// TwinCAT 3 PLC project OP710_Robotic_Weld
// ProgramVersion: 3.1.4024.0
// libraries:
//   Tc2_Standard, * (Beckhoff Automation GmbH)
//   Tc2_System, * (Beckhoff Automation GmbH)
//   Tc3_Module, * (Beckhoff Automation GmbH)
//   VisuDialogs, * (System)
// project tree:
//   DUTs/ Fixture.TcDUT, MH_Robot.TcDUT, Weld_Robot.TcDUT
//   / GlobalTextList.TcGTLO, PlcTask.TcTTO, Visualization Manager.TcVMO (not stored)
//   GVLs/ Inputs.TcGVL, Memory.TcGVL, Outputs.TcGVL
//   POUs/ Auto_Cycle_Fix1.TcPOU, Auto_Cycle_Fix2.TcPOU, Fix1_FB.TcPOU, Fix2_FB.TcPOU, MAIN.TcPOU, Robot_MH.TcPOU, Robot_Weld.TcPOU, RollerDoor.TcPOU, Trunnion.TcPOU, TurnTable.TcPOU
//   VISUs/ Auto_Cycle_Fix1.TcVIS, Auto_Cycle_Fix2.TcVIS, Manual_Action_Fix1.TcVIS, Manual_Action_Fix2.TcVIS
// real-time tasks:
//   TASK PlcTask: cycle T#10ms, priority 20, ADS port 350

CONFIGURATION OP710_Robotic_Weld
    RESOURCE PLC ON TwinCAT3
        TASK PlcTask(INTERVAL := T#10ms, PRIORITY := 20);
        PROGRAM MAIN WITH PlcTask : MAIN;
    END_RESOURCE
END_CONFIGURATION

// ---- DUTs/Fixture.TcDUT
TYPE Fixture :
STRUCT
	i_Clamp1_Fbk : BOOL;
	i_Clamp2_Fbk : BOOL;
	i_Clamp3_Fbk : BOOL;
	
	i_Declamp1_Fbk : BOOL;
	i_Declamp2_Fbk : BOOL;
	i_Declamp3_Fbk : BOOL;
	
	o_Clamp_HP : BOOL;
	o_Clamp_WP : BOOL;
	
	Work_Position : BOOL;
	Home_Position : BOOL;
	Manual_Sel : BOOL;
	Auto_Sel : BOOL;
	
END_STRUCT
END_TYPE

// ---- DUTs/MH_Robot.TcDUT
TYPE MH_Robot :
STRUCT
	i_Home 			: BOOL;
	i_Prg_No		: INT;
	i_Start			: BOOL;	
	i_Area_Ok1		: BOOL;
	i_Area_Ok2		: BOOL;
	
	o_Pickup_Comp1	: BOOL;
	o_Pickup_Comp2	: BOOL;
		
END_STRUCT
END_TYPE

// ---- DUTs/Weld_Robot.TcDUT
TYPE Weld_Robot :
STRUCT
	i_Home 		: BOOL;
	i_Prg_No	: INT;
	i_Start		: BOOL;	
	i_Area_Ok	: BOOL;
	
	o_Weld_Comp	: BOOL;
	
END_STRUCT
END_TYPE

// ---- GVLs/Inputs.TcGVL

//(------INPUTS--------)

VAR_GLOBAL
	
i_Control_Pressure_Sw_In1_BPB1 AT %IX0.0 : BOOL;	//Control Pressure Switch Input 1-BPB1  
i_Control_Pressure_Sw_In2_BPB1 AT %IX0.1 : BOOL;	//Control Pressure Switch Input 2-BPB1  
i_Valve_Pos_BGB1 AT %IX0.2 : BOOL;					//Valve Position-BGB1
i_CC6_Clamp_1_Sensor_HP AT %IX0.4 : BOOL;			//Clamping Circuit 6 Clamping Unit 1 sensor  HP
i_CC6_Clamp_1_Sensor_WP AT %IX0.5 : BOOL;			//Clamping Circuit 6 Clamping Unit 1 sensor  WP
i_CC4_Clamp_3_Sensor_HP AT %IX0.6 : BOOL;			//Clamping Circuit 4 Clamping Unit 3 sensor  HP
i_CC4_Clamp_3_Sensor_WP AT %IX0.7 : BOOL;			//Clamping Circuit 4 Clamping Unit 3 sensor  WP
i_PART_CONTROL_B13 AT %IX1.0 : BOOL;				//PART CONTROL  B13
i_PART_CONTROL_B27 AT %IX1.1 : BOOL;				//PART CONTROL  B27
i_PART_CONTROL_B14 AT %IX1.2 : BOOL;				//PART CONTROL  B14
i_PART_CONTROL_B28 AT %IX1.3 : BOOL;				//PART CONTROL  B28
i_KEC6_Slave_module_1_2_1 AT %IX1.6 : BOOL;			//Connect to KEC6 Salve module 1.2
i_KEC6_Slave_module_1_2_2 AT %IX1.7 : BOOL;			//Connect to KEC6 Salve module 1.2

i_CC4_Clamp_2_Sensor_HP	AT %IX4.0 : BOOL;			//Clamping Circuit 4 Clamping Unit 2 sensor HP
i_CC4_Clamp_2_Sensor_WP	AT %IX4.1 : BOOL;			//Clamping Circuit 4 Clamping Unit 2 sensor WP
i_CC4_Clamp_1_Sensor_HP	AT %IX4.2 : BOOL;			//Clamping Circuit 4 Clamping Unit 1 sensor HP
i_CC4_Clamp_1_Sensor_WP	AT %IX4.3 : BOOL;			//Clamping Circuit 4 Clamping Unit 1 sensor WP
i_CC2_Clamp_3_Sensor_HP	AT %IX4.4 : BOOL;			//Clamping Circuit 2 Clamping Unit 3 sensor HP
i_CC2_Clamp_3_Sensor_WP	AT %IX4.5 : BOOL;			//Clamping Circuit 2 Clamping Unit 3 sensor WP
i_PART_CONTROL_B12	AT %IX4.6 : BOOL;				//PART CONTROL B12
i_PART_CONTROL_B26	AT %IX4.7 : BOOL;				//PART CONTROL B26

i_PART_CONTROL_B11	AT %IX5.0 : BOOL;				//PART CONTROL B11
i_PART_CONTROL_B25	AT %IX5.1 : BOOL;				//PART CONTROL B25
i_PART_CONTROL_B10	AT %IX5.2 : BOOL;				//PART CONTROL B10
i_PART_CONTROL_B24	AT %IX5.3 : BOOL;				//PART CONTROL B24

i_CC3_Clamp_3_Sensor_HP AT %IX8.0 : BOOL;			//Clamping Circuit 3 Clamping Unit 3 sensor HP
i_CC3_Clamp_3_Sensor_WP AT %IX8.1 : BOOL;			//Clamping Circuit 3 Clamping Unit 3 sensor WP
i_CC3_Clamp_2_Sensor_HP AT %IX8.2 : BOOL;			//Clamping Circuit 3 Clamping Unit 2 sensor HP
i_CC3_Clamp_2_Sensor_WP AT %IX8.3 : BOOL;			//Clamping Circuit 3 Clamping Unit 2 sensor WP
i_CC3_Clamp_1_Sensor_HP AT %IX8.4 : BOOL;			//Clamping Circuit 3 Clamping Unit 1 sensor HP
i_CC3_Clamp_1_Sensor_WP AT %IX8.5 : BOOL;			//Clamping Circuit 3 Clamping Unit 1 sensor WP
i_PART_CONTROL_B7 AT %IX8.6 : BOOL;					//PART CONTROL B7
i_PART_CONTROL_B21 AT %IX8.7 : BOOL;				//PART CONTROL B21

i_PART_CONTROL_B6 AT %IX9.0 : BOOL;					//PART CONTROL B6
i_PART_CONTROL_B20 AT %IX9.1 : BOOL;				//PART CONTROL B20
i_PART_CONTROL_B5 AT %IX9.2 : BOOL;					//PART CONTROL B5
i_PART_CONTROL_B19 AT %IX9.3 : BOOL;				//PART CONTROL B19
i_KEC8_Slave_module_2_2_1 AT %IX9.6 : BOOL;			//Connect to KEC8 Salve module 2.2
i_KEC8_Slave_module_2_2_2 AT %IX9.7 : BOOL;			//Connect to KEC8 Salve module 2.2

i_CC1_Clamp_3_Sensor_HP AT %IX12.0 : BOOL;			//Clamping Circuit 1 Clamping Unit 3 sensor HP
i_CC1_Clamp_3_Sensor_WP AT %IX12.1 : BOOL;			//Clamping Circuit 1 Clamping Unit 3 sensor WP
i_CC1_Clamp_2_Sensor_HP AT %IX12.2 : BOOL;			//Clamping Circuit 1 Clamping Unit 2 sensor HP
i_CC1_Clamp_2_Sensor_WP AT %IX12.3 : BOOL;			//Clamping Circuit 1 Clamping Unit 2 sensor WP
i_CC1_Clamp_1_Sensor_HP AT %IX12.4 : BOOL;			//Clamping Circuit 1 Clamping Unit 1 sensor HP
i_CC1_Clamp_1_Sensor_WP AT %IX12.5 : BOOL;			//Clamping Circuit 1 Clamping Unit 1 sensor WP
i_PART_CONTROL_B4 AT %IX12.6 : BOOL;				//PART CONTROL B4
i_PART_CONTROL_B18 AT %IX12.7 : BOOL;				//PART CONTROL B18

i_PART_CONTROL_B3 AT %IX13.0 : BOOL;				//PART CONTROL B3
i_PART_CONTROL_B17 AT %IX13.1 : BOOL;				//PART CONTROL B17
i_PART_CONTROL_B2 AT %IX13.2 : BOOL;				//PART CONTROL B2
i_PART_CONTROL_B16 AT %IX13.3 : BOOL;				//PART CONTROL B16

i_CC2_Clamp_2_Sensor_HP AT %IX16.0 : BOOL;			//Clamping Circuit 2 Clamping Unit 2 sensor HP
i_CC2_Clamp_2_Sensor_WP AT %IX16.1 : BOOL;			//Clamping Circuit 2 Clamping Unit 2 sensor WP
i_CC2_Clamp_1_Sensor_HP AT %IX16.2 : BOOL;			//Clamping Circuit 2 Clamping Unit 1 sensor HP
i_CC2_Clamp_1_Sensor_WP AT %IX16.3 : BOOL;			//Clamping Circuit 2 Clamping Unit 1 sensor WP
i_PART_CONTROL_B9 AT %IX16.4 : BOOL;				//PART CONTROL B9
i_PART_CONTROL_B23 AT %IX16.5 : BOOL;				//PART CONTROL B23
i_PART_CONTROL_B8 AT %IX16.6 : BOOL;				//PART CONTROL B8
i_PART_CONTROL_B22 AT %IX16.7 : BOOL;				//PART CONTROL B22

i_CC5_Clamp_1_Sensor_HP AT %IX24.0 : BOOL;			//Clamping Circuit 5 Clamping Unit 1 sensor HP
i_CC5_Clamp_1_Sensor_WP AT %IX24.1 : BOOL;			//Clamping Circuit 5 Clamping Unit 1 sensor WP
i_PART_CONTROL_B1 AT %IX24.2 : BOOL;				//PART CONTROL B1
i_PART_CONTROL_B15 AT %IX24.3 : BOOL;				//PART CONTROL B15

i_TR_0_Deg AT %I* : BOOL;							//Trunnion at 0 degree
i_TR_20_Degree AT %I* : BOOL;						//Trunnion at -20 degree
i_TR_45_Degree AT %I* : BOOL;						//Trunnion at 45 degree
i_TR_50_Degree AT %I* : BOOL;						//Trunnion at 50 degree
i_TR_80_Degree AT %I* : BOOL;						//Trunnion at 80 degree
i_TT_0_Degree AT %I* : BOOL;
i_TT_180_Degree AT %I* : BOOL;

Roller_Door_Up AT %I* : BOOL;						//Roller Door Up
Roller_Door_Down AT %I* : BOOL;						//Roller Door Down


END_VAR

// ---- GVLs/Memory.TcGVL
VAR_GLOBAL
	
Start_Pb     		: BOOL;						    // Station Cycle Start Pb
Station_Mode 		: INT;							// Station Manual/Auto Pb
Fix_Sel   	 		: INT;							//Station Select Pb, 0 - OP710 Long, 1 - OP710 Short
Auto_Mode	 		: BOOL;
Manual_Mode	 		: BOOL;
Master_On	 		: BOOL;
EStop				: BOOL;
Safety_Ok	 		: BOOL;
Fault_Reset			: BOOL;
Fix1_Part_1_Load  	: BOOL;
Fix1_Part_2_Load  	: BOOL;
Fix2_Part_1_Load  	: BOOL;
Fix2_Part_2_Load  	: BOOL;
Return_Home  		: BOOL;

i_B : ARRAY [0..28] OF BOOL;						// Part Sensor Load

END_VAR

// ---- GVLs/Outputs.TcGVL

//(------OUTPUTS--------)

VAR_GLOBAL
	
o_CC1_CLAMPING_UNIT1_3_WP AT %QX0.0 : BOOL;		//Clamping Circuit 1 Clamping Unit 1-3 WP
o_CC1_CLAMPING_UNIT1_3_HP AT %QX0.1 : BOOL;		//Clamping Circuit 1 Clamping Unit 1-3 HP
o_CC2_CLAMPING_UNIT1_3_WP AT %QX0.2 : BOOL;		//Clamping Circuit 2 Clamping Unit 1-3 WP
o_CC2_CLAMPING_UNIT1_3_HP AT %QX0.3 : BOOL;		//Clamping Circuit 2 Clamping Unit 1-3 HP
o_CC3_CLAMPING_UNIT1_3_WP AT %QX0.4 : BOOL;		//Clamping Circuit 3 Clamping Unit 1-3 WP
o_CC3_CLAMPING_UNIT1_3_HP AT %QX0.5 : BOOL;		//Clamping Circuit 3 Clamping Unit 1-3 HP
o_CC4_CLAMPING_UNIT1_3_WP AT %QX0.6 : BOOL;		//Clamping Circuit 4 Clamping Unit 1-3 WP
o_CC4_CLAMPING_UNIT1_3_HP AT %QX0.7 : BOOL;		//Clamping Circuit 4 Clamping Unit 1-3 HP

o_CC5_CLAMPING_UNIT1_3_WP AT %QX1.0 : BOOL;		//Clamping Circuit 5 Clamping Unit 1 WP
o_CC5_CLAMPING_UNIT1_3_HP AT %QX1.1 : BOOL;		//Clamping Circuit 5 Clamping Unit 1 HP
o_CC6_CLAMPING_UNIT1_3_WP AT %QX1.2 : BOOL;		//Clamping Circuit 6 Clamping Unit 1 WP
o_CC6_CLAMPING_UNIT1_3_HP AT %QX1.3 : BOOL;		//Clamping Circuit 6 Clamping Unit 1 HP

i_TR_0_Deg_Cmd AT %Q* : BOOL;
i_TR_20_Deg_Cmd AT %Q* : BOOL;					//Trunnion at -20 degree
i_TR_45_Deg_Cmd AT %Q* : BOOL;					//Trunnion at 45 degree
i_TR_50_Deg_Cmd AT %Q* : BOOL;					//Trunnion at 50 degree
i_TR_80_Deg_Cmd AT %Q* : BOOL;					//Trunnion at 80 degree
i_TT_0_Deg_Cmd AT %Q* : BOOL;
i_TT_180_Deg_Cmd AT %Q* : BOOL;

Roller_Door_Up_Cmd AT %Q* : BOOL;				//Roller Door Up
Roller_Door_Down_Cmd AT %Q* : BOOL;				//Roller Door Down


END_VAR

// ---- POUs/MAIN.TcPOU
PROGRAM MAIN
VAR
END_VAR

IF Estop THEN
	Safety_Ok := FALSE;
END_IF
IF Fault_Reset THEN
	Safety_Ok := TRUE;
END_IF
IF Safety_Ok THEN
Master_On := TRUE;
END_IF
IF Master_On THEN
Auto_Cycle_Fix1();
Auto_Cycle_Fix2();
END_IF

END_PROGRAM

// ---- POUs/Auto_Cycle_Fix1.TcPOU
PROGRAM Auto_Cycle_Fix1
VAR
	Fixture_1 : Fix1_FB;
	TurnTable_0: TurnTable;
	Trunnion_0: Trunnion;
	RollerDoor_0: RollerDoor;
	Robot_Weld_0: Robot_Weld;
	Robot_MH_0: Robot_MH;
END_VAR
VAR // added by the converter: edge detectors and wires of the graphical bodies
    _w1, _w2 : BOOL;
END_VAR

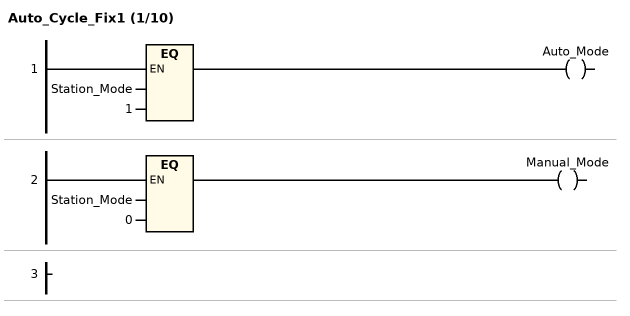
// NETWORK 1
Auto_Mode := Station_Mode = 1;

// NETWORK 2
Manual_Mode := Station_Mode = 0;

// NETWORK 3

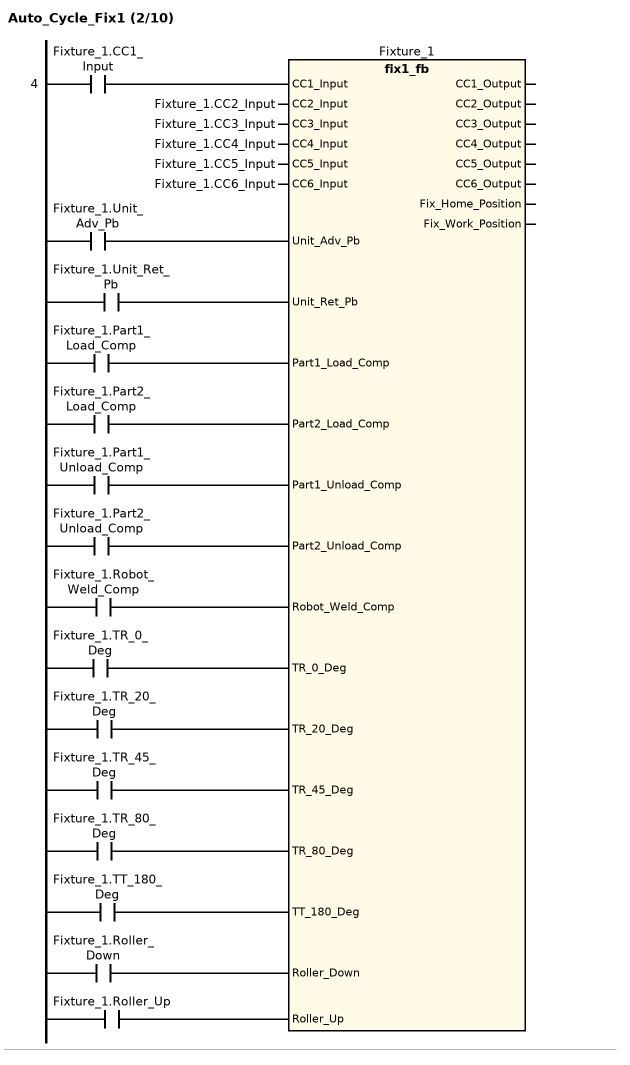
// NETWORK 4
Fixture_1(
    CC1_Input := Fixture_1.CC1_Input,
    CC2_Input := Fixture_1.CC2_Input,
    CC3_Input := Fixture_1.CC3_Input,
    CC4_Input := Fixture_1.CC4_Input,
    CC5_Input := Fixture_1.CC5_Input,
    CC6_Input := Fixture_1.CC6_Input,
    Unit_Adv_Pb := Fixture_1.Unit_Adv_Pb,
    Unit_Ret_Pb := Fixture_1.Unit_Ret_Pb,
    Part1_Load_Comp := Fixture_1.Part1_Load_Comp,
    Part2_Load_Comp := Fixture_1.Part2_Load_Comp,
    Part1_Unload_Comp := Fixture_1.Part1_Unload_Comp,
    Part2_Unload_Comp := Fixture_1.Part2_Unload_Comp,
    Robot_Weld_Comp := Fixture_1.Robot_Weld_Comp,
    TR_0_Deg := Fixture_1.TR_0_Deg,
    TR_20_Deg := Fixture_1.TR_20_Deg,
    TR_45_Deg := Fixture_1.TR_45_Deg,
    TR_80_Deg := Fixture_1.TR_80_Deg,
    TT_180_Deg := Fixture_1.TT_180_Deg,
    Roller_Down := Fixture_1.Roller_Down,
    Roller_Up := Fixture_1.Roller_Up); // fix1_fb

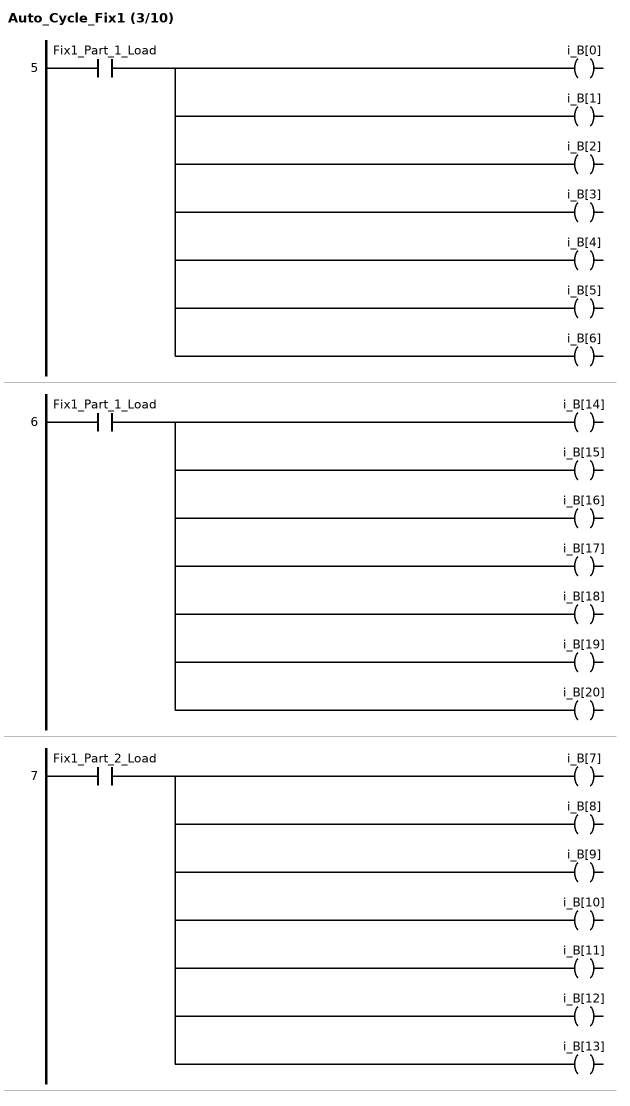
// NETWORK 5
i_B[0] := Fix1_Part_1_Load;
i_B[1] := Fix1_Part_1_Load;
i_B[2] := Fix1_Part_1_Load;
i_B[3] := Fix1_Part_1_Load;
i_B[4] := Fix1_Part_1_Load;
i_B[5] := Fix1_Part_1_Load;
i_B[6] := Fix1_Part_1_Load;

// NETWORK 6
i_B[14] := Fix1_Part_1_Load;
i_B[15] := Fix1_Part_1_Load;
i_B[16] := Fix1_Part_1_Load;
i_B[17] := Fix1_Part_1_Load;
i_B[18] := Fix1_Part_1_Load;
i_B[19] := Fix1_Part_1_Load;
i_B[20] := Fix1_Part_1_Load;

// NETWORK 7
i_B[7] := Fix1_Part_2_Load;
i_B[8] := Fix1_Part_2_Load;
i_B[9] := Fix1_Part_2_Load;
i_B[10] := Fix1_Part_2_Load;
i_B[11] := Fix1_Part_2_Load;
i_B[12] := Fix1_Part_2_Load;
i_B[13] := Fix1_Part_2_Load;

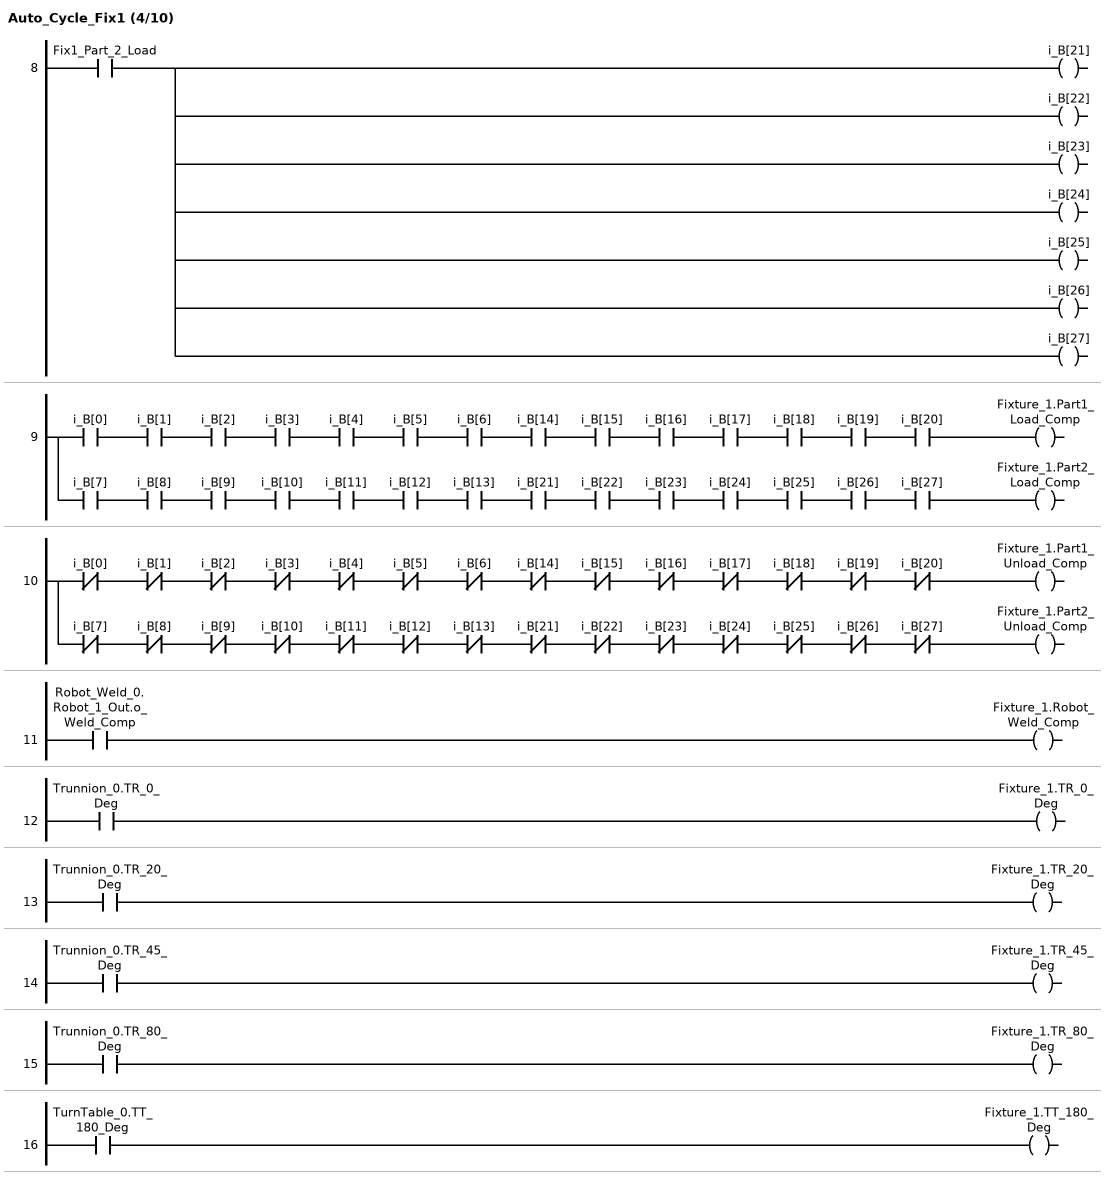
// NETWORK 8
i_B[21] := Fix1_Part_2_Load;
i_B[22] := Fix1_Part_2_Load;
i_B[23] := Fix1_Part_2_Load;
i_B[24] := Fix1_Part_2_Load;
i_B[25] := Fix1_Part_2_Load;
i_B[26] := Fix1_Part_2_Load;
i_B[27] := Fix1_Part_2_Load;

// NETWORK 9
Fixture_1.Part1_Load_Comp := i_B[0] AND i_B[1] AND i_B[2] AND i_B[3] AND i_B[4] AND i_B[5] AND i_B[6] AND i_B[14] AND i_B[15] AND i_B[16] AND i_B[17] AND i_B[18] AND i_B[19] AND i_B[20];
Fixture_1.Part2_Load_Comp := i_B[7] AND i_B[8] AND i_B[9] AND i_B[10] AND i_B[11] AND i_B[12] AND i_B[13] AND i_B[21] AND i_B[22] AND i_B[23] AND i_B[24] AND i_B[25] AND i_B[26] AND i_B[27];

// NETWORK 10
Fixture_1.Part1_Unload_Comp := NOT i_B[0] AND NOT i_B[1] AND NOT i_B[2] AND NOT i_B[3] AND NOT i_B[4] AND NOT i_B[5] AND NOT i_B[6] AND NOT i_B[14] AND NOT i_B[15] AND NOT i_B[16] AND NOT i_B[17] AND NOT i_B[18] AND NOT i_B[19] AND NOT i_B[20];
Fixture_1.Part2_Unload_Comp := NOT i_B[7] AND NOT i_B[8] AND NOT i_B[9] AND NOT i_B[10] AND NOT i_B[11] AND NOT i_B[12] AND NOT i_B[13] AND NOT i_B[21] AND NOT i_B[22] AND NOT i_B[23] AND NOT i_B[24] AND NOT i_B[25] AND NOT i_B[26] AND NOT i_B[27];

// NETWORK 11
Fixture_1.Robot_Weld_Comp := Robot_Weld_0.Robot_1_Out.o_Weld_Comp;

// NETWORK 12
Fixture_1.TR_0_Deg := Trunnion_0.TR_0_Deg;

// NETWORK 13
Fixture_1.TR_20_Deg := Trunnion_0.TR_20_Deg;

// NETWORK 14
Fixture_1.TR_45_Deg := Trunnion_0.TR_45_Deg;

// NETWORK 15
Fixture_1.TR_80_Deg := Trunnion_0.TR_80_Deg;

// NETWORK 16
Fixture_1.TT_180_Deg := TurnTable_0.TT_180_Deg;

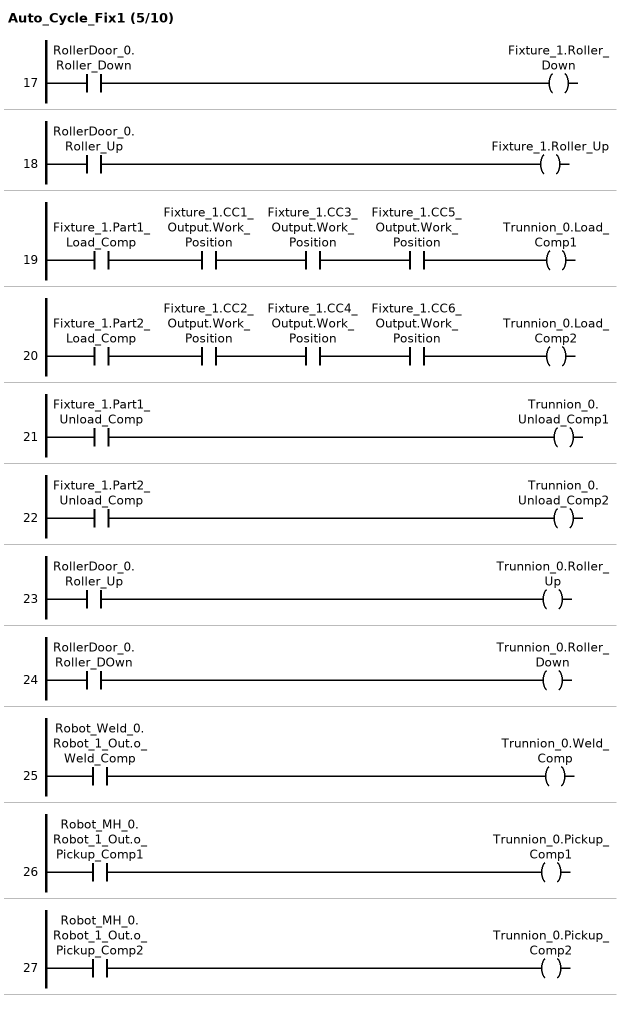
// NETWORK 17
Fixture_1.Roller_Down := RollerDoor_0.Roller_Down;

// NETWORK 18
Fixture_1.Roller_Up := RollerDoor_0.Roller_Up;

// NETWORK 19
Trunnion_0.Load_Comp1 := Fixture_1.Part1_Load_Comp AND Fixture_1.CC1_Output.Work_Position AND Fixture_1.CC3_Output.Work_Position AND Fixture_1.CC5_Output.Work_Position;

// NETWORK 20
Trunnion_0.Load_Comp2 := Fixture_1.Part2_Load_Comp AND Fixture_1.CC2_Output.Work_Position AND Fixture_1.CC4_Output.Work_Position AND Fixture_1.CC6_Output.Work_Position;

// NETWORK 21
Trunnion_0.Unload_Comp1 := Fixture_1.Part1_Unload_Comp;

// NETWORK 22
Trunnion_0.Unload_Comp2 := Fixture_1.Part2_Unload_Comp;

// NETWORK 23
Trunnion_0.Roller_Up := RollerDoor_0.Roller_Up;

// NETWORK 24
Trunnion_0.Roller_Down := RollerDoor_0.Roller_DOwn;

// NETWORK 25
Trunnion_0.Weld_Comp := Robot_Weld_0.Robot_1_Out.o_Weld_Comp;

// NETWORK 26
Trunnion_0.Pickup_Comp1 := Robot_MH_0.Robot_1_Out.o_Pickup_Comp1;

// NETWORK 27
Trunnion_0.Pickup_Comp2 := Robot_MH_0.Robot_1_Out.o_Pickup_Comp2;

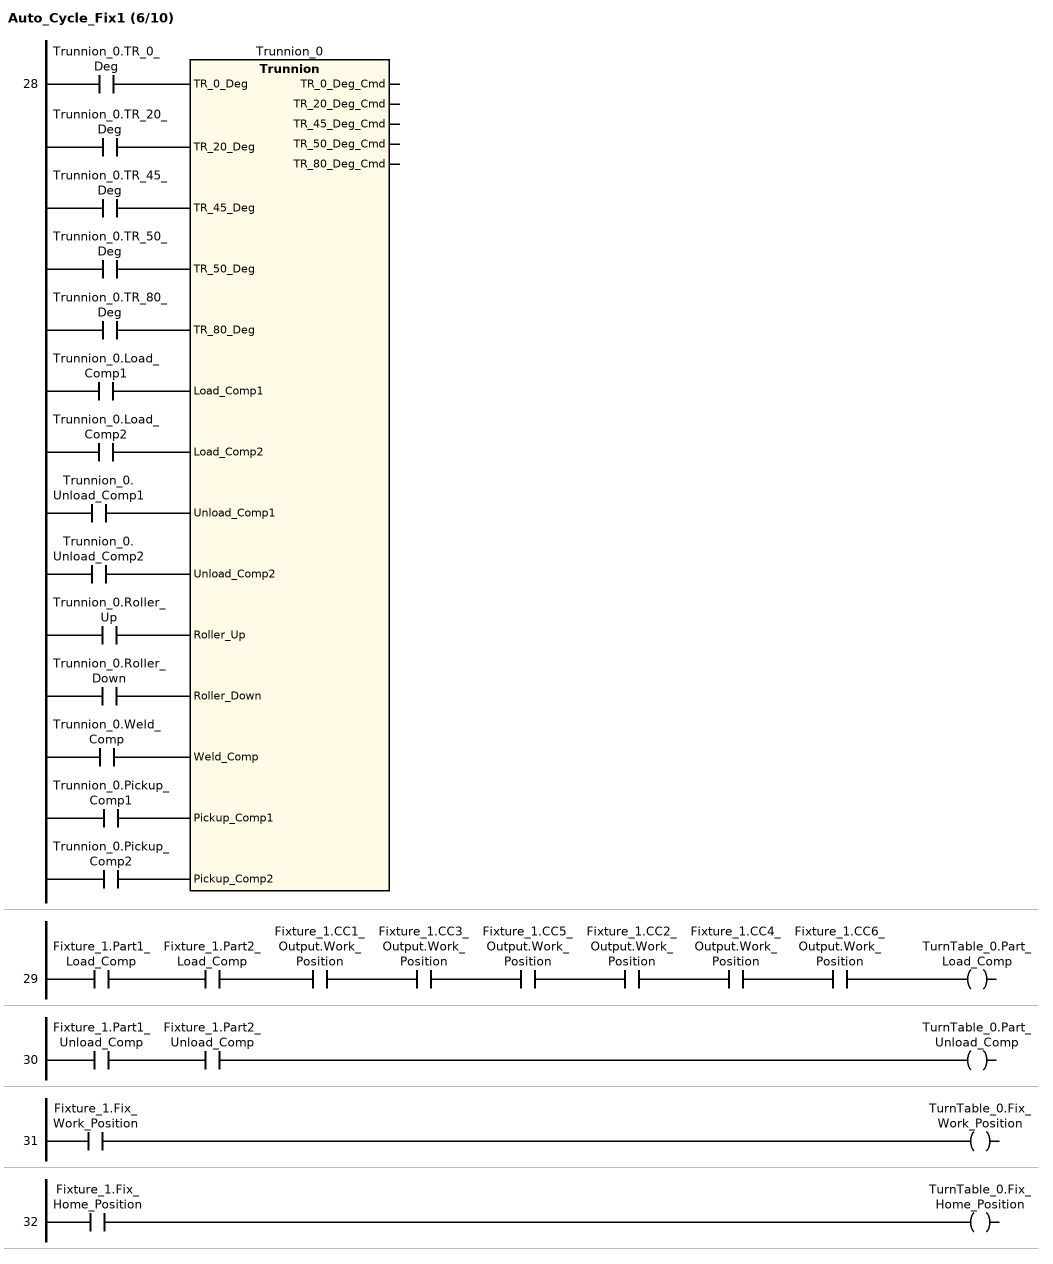
// NETWORK 28
Trunnion_0(
    TR_0_Deg := Trunnion_0.TR_0_Deg,
    TR_20_Deg := Trunnion_0.TR_20_Deg,
    TR_45_Deg := Trunnion_0.TR_45_Deg,
    TR_50_Deg := Trunnion_0.TR_50_Deg,
    TR_80_Deg := Trunnion_0.TR_80_Deg,
    Load_Comp1 := Trunnion_0.Load_Comp1,
    Load_Comp2 := Trunnion_0.Load_Comp2,
    Unload_Comp1 := Trunnion_0.Unload_Comp1,
    Unload_Comp2 := Trunnion_0.Unload_Comp2,
    Roller_Up := Trunnion_0.Roller_Up,
    Roller_Down := Trunnion_0.Roller_Down,
    Weld_Comp := Trunnion_0.Weld_Comp,
    Pickup_Comp1 := Trunnion_0.Pickup_Comp1,
    Pickup_Comp2 := Trunnion_0.Pickup_Comp2); // Trunnion

// NETWORK 29
TurnTable_0.Part_Load_Comp := Fixture_1.Part1_Load_Comp AND Fixture_1.Part2_Load_Comp AND Fixture_1.CC1_Output.Work_Position AND Fixture_1.CC3_Output.Work_Position AND Fixture_1.CC5_Output.Work_Position AND Fixture_1.CC2_Output.Work_Position AND Fixture_1.CC4_Output.Work_Position AND Fixture_1.CC6_Output.Work_Position;

// NETWORK 30
TurnTable_0.Part_Unload_Comp := Fixture_1.Part1_Unload_Comp AND Fixture_1.Part2_Unload_Comp;

// NETWORK 31
TurnTable_0.Fix_Work_Position := Fixture_1.Fix_Work_Position;

// NETWORK 32
TurnTable_0.Fix_Home_Position := Fixture_1.Fix_Home_Position;

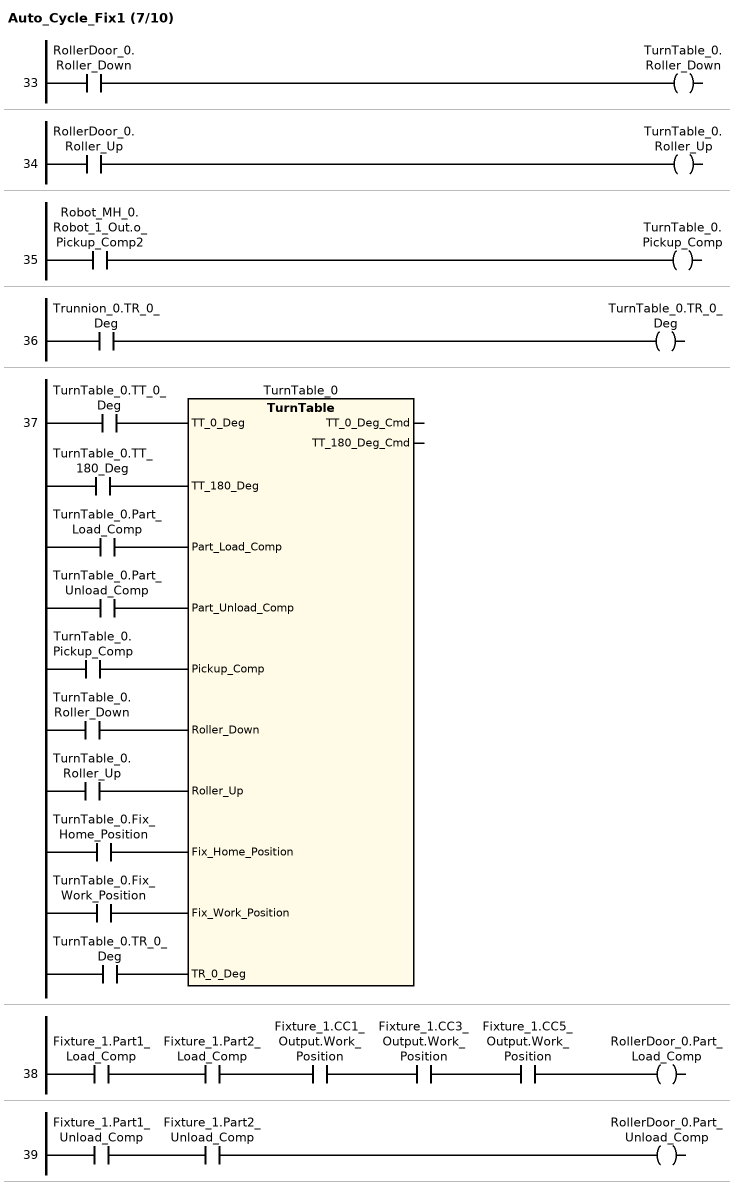
// NETWORK 33
TurnTable_0.Roller_Down := RollerDoor_0.Roller_Down;

// NETWORK 34
TurnTable_0.Roller_Up := RollerDoor_0.Roller_Up;

// NETWORK 35
TurnTable_0.Pickup_Comp := Robot_MH_0.Robot_1_Out.o_Pickup_Comp2;

// NETWORK 36
TurnTable_0.TR_0_Deg := Trunnion_0.TR_0_Deg;

// NETWORK 37
TurnTable_0(
    TT_0_Deg := TurnTable_0.TT_0_Deg,
    TT_180_Deg := TurnTable_0.TT_180_Deg,
    Part_Load_Comp := TurnTable_0.Part_Load_Comp,
    Part_Unload_Comp := TurnTable_0.Part_Unload_Comp,
    Pickup_Comp := TurnTable_0.Pickup_Comp,
    Roller_Down := TurnTable_0.Roller_Down,
    Roller_Up := TurnTable_0.Roller_Up,
    Fix_Home_Position := TurnTable_0.Fix_Home_Position,
    Fix_Work_Position := TurnTable_0.Fix_Work_Position,
    TR_0_Deg := TurnTable_0.TR_0_Deg); // TurnTable

// NETWORK 38
RollerDoor_0.Part_Load_Comp := Fixture_1.Part1_Load_Comp AND Fixture_1.Part2_Load_Comp AND Fixture_1.CC1_Output.Work_Position AND Fixture_1.CC3_Output.Work_Position AND Fixture_1.CC5_Output.Work_Position;

// NETWORK 39
RollerDoor_0.Part_Unload_Comp := Fixture_1.Part1_Unload_Comp AND Fixture_1.Part2_Unload_Comp;

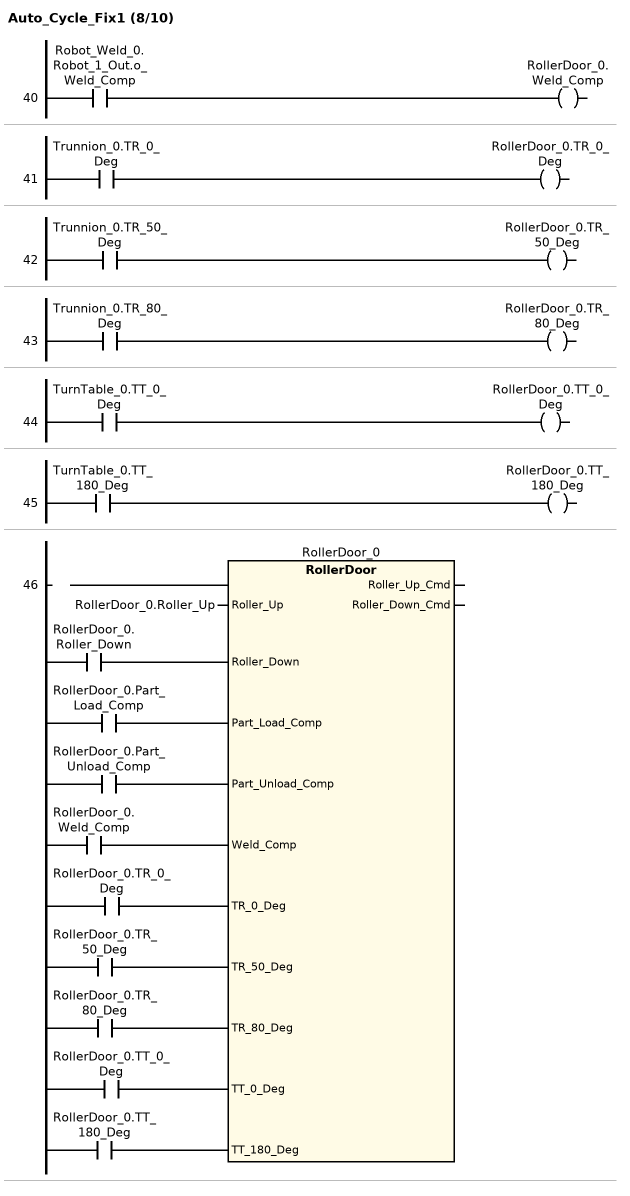
// NETWORK 40
RollerDoor_0.Weld_Comp := Robot_Weld_0.Robot_1_Out.o_Weld_Comp;

// NETWORK 41
RollerDoor_0.TR_0_Deg := Trunnion_0.TR_0_Deg;

// NETWORK 42
RollerDoor_0.TR_50_Deg := Trunnion_0.TR_50_Deg;

// NETWORK 43
RollerDoor_0.TR_80_Deg := Trunnion_0.TR_80_Deg;

// NETWORK 44
RollerDoor_0.TT_0_Deg := TurnTable_0.TT_0_Deg;

// NETWORK 45
RollerDoor_0.TT_180_Deg := TurnTable_0.TT_180_Deg;

// NETWORK 46
RollerDoor_0(
    Roller_Up := RollerDoor_0.Roller_Up,
    Roller_Down := RollerDoor_0.Roller_Down,
    Part_Load_Comp := RollerDoor_0.Part_Load_Comp,
    Part_Unload_Comp := RollerDoor_0.Part_Unload_Comp,
    Weld_Comp := RollerDoor_0.Weld_Comp,
    TR_0_Deg := RollerDoor_0.TR_0_Deg,
    TR_50_Deg := RollerDoor_0.TR_50_Deg,
    TR_80_Deg := RollerDoor_0.TR_80_Deg,
    TT_0_Deg := RollerDoor_0.TT_0_Deg,
    TT_180_Deg := RollerDoor_0.TT_180_Deg); // RollerDoor

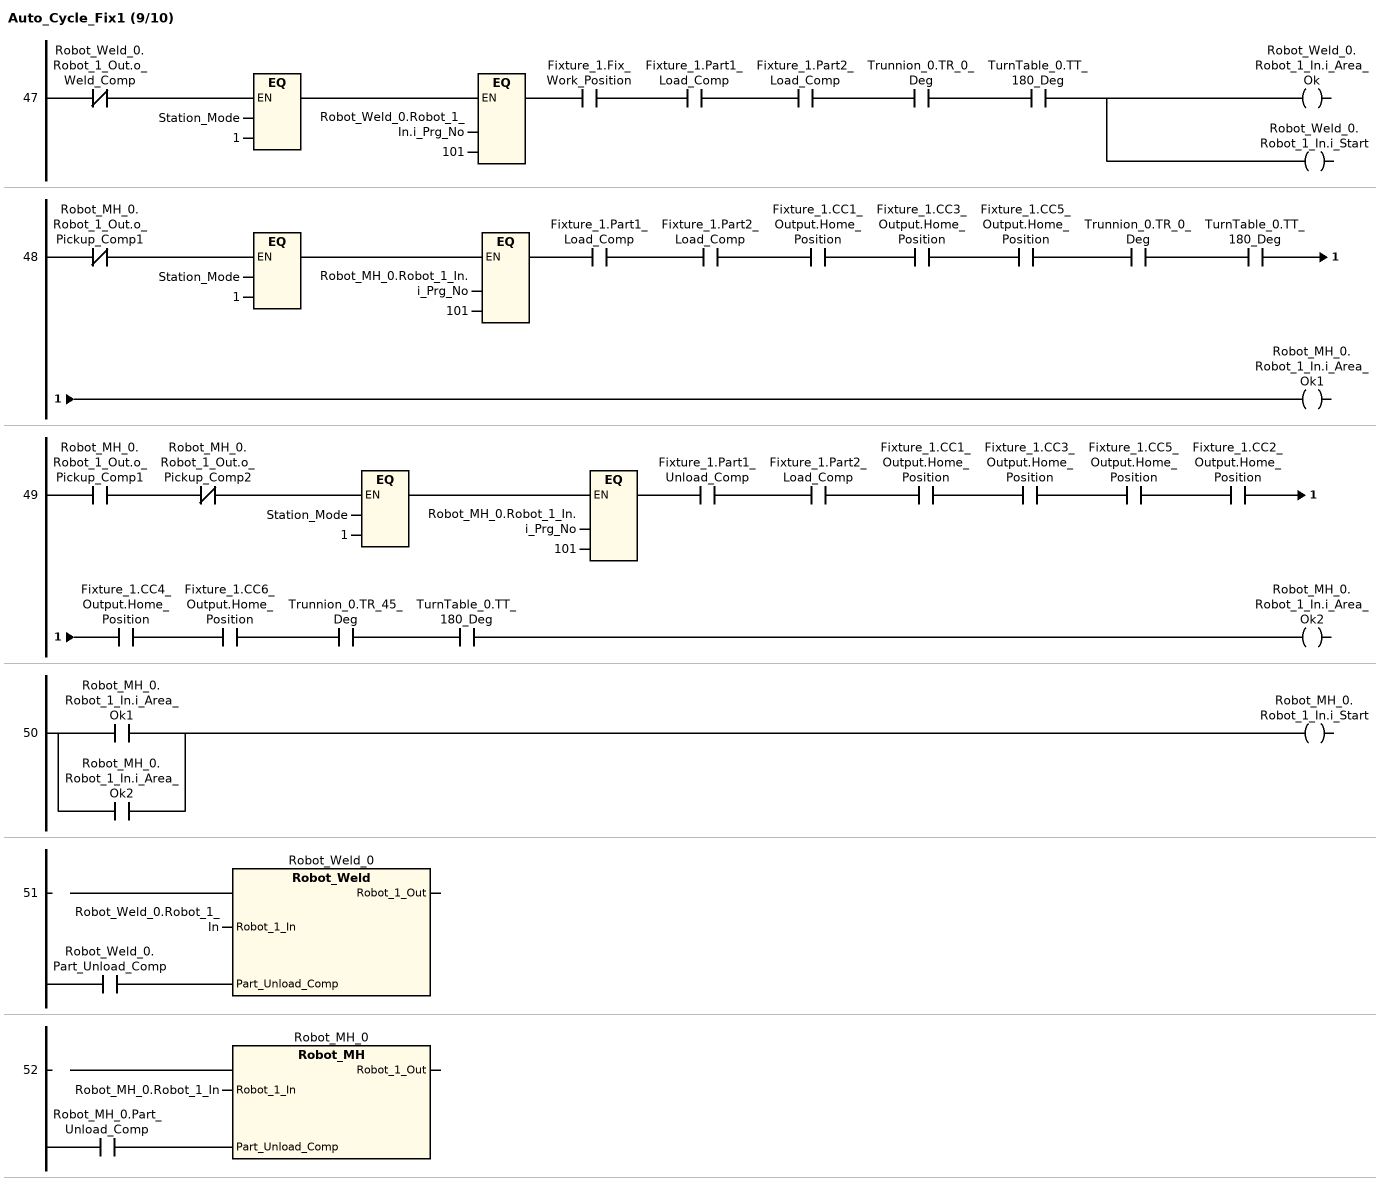
// NETWORK 47
_w1 := (NOT Robot_Weld_0.Robot_1_Out.o_Weld_Comp AND Station_Mode = 1 AND Robot_Weld_0.Robot_1_In.i_Prg_No = 101) AND Fixture_1.Fix_Work_Position AND Fixture_1.Part1_Load_Comp AND Fixture_1.Part2_Load_Comp AND Trunnion_0.TR_0_Deg AND TurnTable_0.TT_180_Deg;
Robot_Weld_0.Robot_1_In.i_Area_Ok := _w1;
Robot_Weld_0.Robot_1_In.i_Start := _w1;

// NETWORK 48
Robot_MH_0.Robot_1_In.i_Area_Ok1 := (NOT Robot_MH_0.Robot_1_Out.o_Pickup_Comp1 AND Station_Mode = 1 AND Robot_MH_0.Robot_1_In.i_Prg_No = 101) AND Fixture_1.Part1_Load_Comp AND Fixture_1.Part2_Load_Comp AND Fixture_1.CC1_Output.Home_Position AND Fixture_1.CC3_Output.Home_Position AND Fixture_1.CC5_Output.Home_Position AND Trunnion_0.TR_0_Deg AND TurnTable_0.TT_180_Deg;

// NETWORK 49
Robot_MH_0.Robot_1_In.i_Area_Ok2 := (Robot_MH_0.Robot_1_Out.o_Pickup_Comp1 AND NOT Robot_MH_0.Robot_1_Out.o_Pickup_Comp2 AND Station_Mode = 1 AND Robot_MH_0.Robot_1_In.i_Prg_No = 101) AND Fixture_1.Part1_Unload_Comp AND Fixture_1.Part2_Load_Comp AND Fixture_1.CC1_Output.Home_Position AND Fixture_1.CC3_Output.Home_Position AND Fixture_1.CC5_Output.Home_Position AND Fixture_1.CC2_Output.Home_Position AND Fixture_1.CC4_Output.Home_Position AND Fixture_1.CC6_Output.Home_Position AND Trunnion_0.TR_45_Deg AND TurnTable_0.TT_180_Deg;

// NETWORK 50
Robot_MH_0.Robot_1_In.i_Start := Robot_MH_0.Robot_1_In.i_Area_Ok1 OR Robot_MH_0.Robot_1_In.i_Area_Ok2;

// NETWORK 51
Robot_Weld_0(Robot_1_In := Robot_Weld_0.Robot_1_In, Part_Unload_Comp := Robot_Weld_0.Part_Unload_Comp); // Robot_Weld

// NETWORK 52
Robot_MH_0(Robot_1_In := Robot_MH_0.Robot_1_In, Part_Unload_Comp := Robot_MH_0.Part_Unload_Comp); // Robot_MH

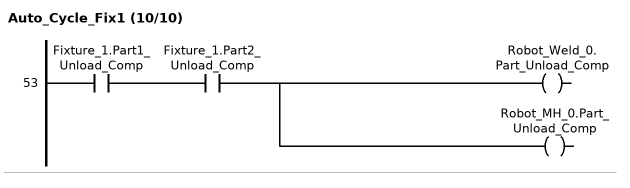
// NETWORK 53
_w2 := Fixture_1.Part1_Unload_Comp AND Fixture_1.Part2_Unload_Comp;
Robot_Weld_0.Part_Unload_Comp := _w2;
Robot_MH_0.Part_Unload_Comp := _w2;

END_PROGRAM

// ---- POUs/Fix1_FB.TcPOU
FUNCTION_BLOCK Fix1_FB
VAR_INPUT
CC1_Input 			: Fixture;					//Clamping Circuit-1
CC2_Input 			: Fixture;					//Clamping Circuit-2
CC3_Input 			: Fixture;					//Clamping Circuit-3
CC4_Input 			: Fixture;					//Clamping Circuit-4
CC5_Input 			: Fixture;					//Clamping Circuit-5
CC6_Input 			: Fixture;					//Clamping Circuit-6

Unit_Adv_Pb 		: BOOL;						//Fixture Cylinder Clamp Pb
Unit_Ret_Pb 		: BOOL;						//Fixture Cylinder Declamp Pb

Part1_Load_Comp 	: BOOL;						//OP710 Part-1 Load Complete
Part2_Load_Comp 	: BOOL;						//OP710 Part-2 Load Complete
Part1_Unload_Comp 	: BOOL;						//OP710 Part-1 Unload Complete
Part2_Unload_Comp 	: BOOL;						//OP710 Part-2 Unload Complete

Robot_Weld_Comp 	: BOOL;						//Robot Weld Complete
TR_0_Deg  			: BOOL;						//Trunnion at 0 degree
TR_20_Deg 			: BOOL;						//Trunnion at -20 degree
TR_45_Deg 			: BOOL;						//Trunnion at 45 degree
TR_80_Deg 			: BOOL;						//Trunnion at 80 degree

TT_180_Deg 		: BOOL;						//Trunnion at 180 degree
Roller_Down 		: BOOL;						//Roller Door Down position
Roller_Up 			: BOOL;						//Roller Door Up position
END_VAR

VAR_OUTPUT
CC1_Output 			: Fixture;							//Clamping Circuit-1
CC2_Output 			: Fixture;							//Clamping Circuit-2
CC3_Output 			: Fixture;							//Clamping Circuit-3
CC4_Output 			: Fixture;							//Clamping Circuit-4
CC5_Output 			: Fixture;							//Clamping Circuit-5
CC6_Output 			: Fixture;							//Clamping Circuit-6
Fix_Home_Position 	: BOOL;
Fix_Work_Position 	: BOOL;

END_VAR

VAR
Cyl_Delay 			: ARRAY [0..30] OF TON;
END_VAR

Fix_Home_Position := CC1_Output.Home_Position AND CC2_Output.Home_Position AND CC3_Output.Home_Position AND CC4_Output.Home_Position AND CC5_Output.Home_Position AND CC6_Output.Home_Position;
Fix_Work_Position := CC1_Output.Work_Position AND CC2_Output.Work_Position AND CC3_Output.Work_Position AND CC4_Output.Work_Position AND CC5_Output.Work_Position AND CC6_Output.Work_Position;

CASE Station_Mode OF
	
	0: 
	
	IF (CC1_Input.Manual_Sel AND Unit_Adv_Pb AND (NOT Unit_Ret_Pb) AND CC3_Output.Home_Position) THEN
		CC1_Output.o_Clamp_WP := TRUE;
		Cyl_Delay[0](IN:= CC1_Output.o_Clamp_WP, PT:= T#1S, Q=> , ET=> );
		IF Cyl_Delay[0].Q THEN
		CC1_Input.i_Clamp1_Fbk := CC1_Input.i_Clamp2_Fbk := CC1_Input.i_Clamp3_Fbk := CC1_Output.Work_Position := TRUE;
		CC1_Input.i_Declamp1_Fbk := CC1_Input.i_Declamp2_Fbk := CC1_Input.i_Declamp3_Fbk := CC1_Output.Home_Position := FALSE;
		CC1_Output.o_Clamp_WP := FALSE;
		END_IF
	ELSIF (CC1_Input.Manual_Sel AND Unit_Ret_Pb AND (NOT Unit_Adv_Pb) AND CC3_Output.Home_Position) THEN
		CC1_Output.o_Clamp_HP := TRUE;
		Cyl_Delay[1](IN:= CC1_Output.o_Clamp_HP, PT:= T#1S, Q=> , ET=> );
		IF Cyl_Delay[1].Q THEN
		CC1_Input.i_Declamp1_Fbk := CC1_Input.i_Declamp2_Fbk := CC1_Input.i_Declamp3_Fbk := CC1_Output.Home_Position := TRUE;
		CC1_Input.i_Clamp1_Fbk := CC1_Input.i_Clamp2_Fbk := CC1_Input.i_Clamp3_Fbk := CC1_Output.Work_Position := FALSE;
		CC1_Output.o_Clamp_HP := FALSE;
		END_IF
	END_IF
	
	IF (CC3_Input.Manual_Sel AND Unit_Adv_Pb AND (NOT Unit_Ret_Pb) AND CC1_Output.Work_Position) THEN
		CC3_Output.o_Clamp_WP := TRUE;
		Cyl_Delay[2](IN:= CC3_Output.o_Clamp_WP, PT:= T#1S, Q=> , ET=> );
		IF Cyl_Delay[2].Q THEN
		CC3_Input.i_Clamp1_Fbk := CC3_Input.i_Clamp2_Fbk := CC3_Input.i_Clamp3_Fbk := CC3_Output.Work_Position := TRUE;
		CC3_Input.i_Declamp1_Fbk := CC3_Input.i_Declamp2_Fbk := CC3_Input.i_Declamp3_Fbk := CC3_Output.Home_Position := FALSE;
		CC3_Output.o_Clamp_WP := FALSE;
		END_IF
	ELSIF (CC3_Input.Manual_Sel AND Unit_Ret_Pb AND (NOT Unit_Adv_Pb) AND CC1_Output.Work_Position) THEN
		CC3_Output.o_Clamp_HP := TRUE;
		Cyl_Delay[3](IN:= CC3_Output.o_Clamp_HP, PT:= T#1S, Q=> , ET=> );
		IF Cyl_Delay[3].Q THEN
		CC3_Input.i_Declamp1_Fbk := CC3_Input.i_Declamp2_Fbk := CC3_Input.i_Declamp3_Fbk := CC3_Output.Home_Position := TRUE;
		CC3_Input.i_Clamp1_Fbk := CC3_Input.i_Clamp2_Fbk := CC3_Input.i_Clamp3_Fbk := CC3_Output.Work_Position := FALSE;
		CC3_Output.o_Clamp_HP := FALSE;
		END_IF
	END_IF
	
	IF (CC5_Input.Manual_Sel AND Unit_Adv_Pb AND (NOT Unit_Ret_Pb) AND CC3_Output.Work_Position) THEN
		CC5_Output.o_Clamp_WP := TRUE;
		Cyl_Delay[4](IN:= CC5_Output.o_Clamp_WP, PT:= T#1S, Q=> , ET=> );
		IF Cyl_Delay[4].Q THEN
		CC5_Input.i_Clamp1_Fbk := CC5_Input.i_Clamp2_Fbk := CC5_Input.i_Clamp3_Fbk := CC5_Output.Work_Position := TRUE;
		CC5_Input.i_Declamp1_Fbk := CC5_Input.i_Declamp2_Fbk := CC5_Input.i_Declamp3_Fbk := CC5_Output.Home_Position := FALSE;
		CC5_Output.o_Clamp_WP := FALSE;
		END_IF
	ELSIF (CC5_Input.Manual_Sel AND Unit_Ret_Pb AND (NOT Unit_Adv_Pb) AND CC3_Output.Work_Position) THEN
		CC5_Output.o_Clamp_HP := TRUE;
		Cyl_Delay[5](IN:= CC5_Output.o_Clamp_HP, PT:= T#1S, Q=> , ET=> );
		IF Cyl_Delay[5].Q THEN
		CC5_Input.i_Declamp1_Fbk := CC5_Input.i_Declamp2_Fbk := CC5_Input.i_Declamp3_Fbk := CC5_Output.Home_Position := TRUE;
		CC5_Input.i_Clamp1_Fbk := CC5_Input.i_Clamp2_Fbk := CC5_Input.i_Clamp3_Fbk := CC5_Output.Work_Position := FALSE;
		CC5_Output.o_Clamp_HP := FALSE;
		END_IF
	END_IF
	
	IF (CC2_Input.Manual_Sel AND Unit_Adv_Pb AND (NOT Unit_Ret_Pb) AND CC5_Output.Work_Position) THEN
		CC2_Output.o_Clamp_WP := TRUE;
		Cyl_Delay[6](IN:= CC2_Output.o_Clamp_WP, PT:= T#1S, Q=> , ET=> );
		IF Cyl_Delay[6].Q THEN
		CC2_Input.i_Clamp1_Fbk := CC2_Input.i_Clamp2_Fbk := CC2_Input.i_Clamp3_Fbk := CC2_Output.Work_Position := TRUE;
		CC2_Input.i_Declamp1_Fbk := CC2_Input.i_Declamp2_Fbk := CC2_Input.i_Declamp3_Fbk := CC2_Output.Home_Position := FALSE;
		CC2_Output.o_Clamp_WP := FALSE;
		END_IF
	ELSIF (CC2_Input.Manual_Sel AND Unit_Ret_Pb AND (NOT Unit_Adv_Pb) AND CC5_Output.Work_Position) THEN
		CC2_Output.o_Clamp_HP := TRUE;
		Cyl_Delay[7](IN:= CC2_Output.o_Clamp_HP, PT:= T#1S, Q=> , ET=> );
		IF Cyl_Delay[7].Q THEN
		CC2_Input.i_Declamp1_Fbk := CC2_Input.i_Declamp2_Fbk := CC2_Input.i_Declamp3_Fbk := CC2_Output.Home_Position := TRUE;
		CC2_Input.i_Clamp1_Fbk := CC2_Input.i_Clamp2_Fbk := CC2_Input.i_Clamp3_Fbk := CC2_Output.Work_Position := FALSE;
		CC2_Output.o_Clamp_HP := FALSE;
		END_IF
	END_IF
	
	IF (CC4_Input.Manual_Sel AND Unit_Adv_Pb AND (NOT Unit_Ret_Pb) AND CC2_Output.Work_Position) THEN
		CC4_Output.o_Clamp_WP := TRUE;
		Cyl_Delay[8](IN:= CC4_Output.o_Clamp_WP, PT:= T#1S, Q=> , ET=> );
		IF Cyl_Delay[8].Q THEN
		CC4_Input.i_Clamp1_Fbk := CC4_Input.i_Clamp2_Fbk := CC4_Input.i_Clamp3_Fbk := CC4_Output.Work_Position := TRUE;
		CC4_Input.i_Declamp1_Fbk := CC4_Input.i_Declamp2_Fbk := CC4_Input.i_Declamp3_Fbk := CC4_Output.Home_Position := FALSE;
		CC4_Output.o_Clamp_WP := FALSE;
		END_IF
	ELSIF (CC4_Input.Manual_Sel AND Unit_Ret_Pb AND (NOT Unit_Adv_Pb) AND CC2_Output.Work_Position) THEN
		CC4_Output.o_Clamp_HP := TRUE;
		Cyl_Delay[9](IN:= CC4_Output.o_Clamp_HP, PT:= T#1S, Q=> , ET=> );
		IF Cyl_Delay[9].Q THEN
		CC4_Input.i_Declamp1_Fbk := CC4_Input.i_Declamp2_Fbk := CC4_Input.i_Declamp3_Fbk := CC4_Output.Home_Position := TRUE;
		CC4_Input.i_Clamp1_Fbk := CC4_Input.i_Clamp2_Fbk := CC4_Input.i_Clamp3_Fbk := CC4_Output.Work_Position := FALSE;
		CC4_Output.o_Clamp_HP := FALSE;
		END_IF
	END_IF
	
	IF (CC6_Input.Manual_Sel AND Unit_Adv_Pb AND (NOT Unit_Ret_Pb) AND CC4_Output.Work_Position) THEN
		CC6_Output.o_Clamp_WP := TRUE;
		Cyl_Delay[10](IN:= CC6_Output.o_Clamp_WP, PT:= T#1S, Q=> , ET=> );
		IF Cyl_Delay[10].Q THEN
		CC6_Input.i_Clamp1_Fbk := CC6_Input.i_Clamp2_Fbk := CC6_Input.i_Clamp3_Fbk := CC6_Output.Work_Position := TRUE;
		CC6_Input.i_Declamp1_Fbk := CC6_Input.i_Declamp2_Fbk := CC6_Input.i_Declamp3_Fbk := CC6_Output.Home_Position := FALSE;
		CC6_Output.o_Clamp_WP := FALSE;
		END_IF
	ELSIF (CC6_Input.Manual_Sel AND Unit_Ret_Pb AND (NOT Unit_Adv_Pb) AND CC4_Output.Work_Position) THEN
		CC6_Output.o_Clamp_HP := TRUE;
		Cyl_Delay[11](IN:= CC6_Output.o_Clamp_HP, PT:= T#1S, Q=> , ET=> );
		IF Cyl_Delay[11].Q THEN
		CC6_Input.i_Declamp1_Fbk := CC6_Input.i_Declamp2_Fbk := CC6_Input.i_Declamp3_Fbk := CC6_Output.Home_Position := TRUE;
		CC6_Input.i_Clamp1_Fbk := CC6_Input.i_Clamp2_Fbk := CC6_Input.i_Clamp3_Fbk := CC6_Output.Work_Position := FALSE;
		CC6_Output.o_Clamp_HP := FALSE;
		END_IF
	END_IF

	
	1:

	IF (Start_Pb AND CC1_Input.Auto_Sel AND TR_20_Deg AND Part1_Load_Comp AND CC3_Output.Home_Position) THEN
		CC1_Output.o_Clamp_WP := TRUE;
		Cyl_Delay[12](IN:= (CC1_Output.o_Clamp_WP), PT:= T#1S, Q=> , ET=> );
		IF Cyl_Delay[12].Q THEN
		CC1_Input.i_Declamp1_Fbk := CC1_Input.i_Declamp2_Fbk := CC1_Input.i_Declamp3_Fbk := CC1_Output.Home_Position := FALSE;
		CC1_Input.i_Clamp1_Fbk := CC1_Input.i_Clamp2_Fbk := CC1_Input.i_Clamp3_Fbk := CC1_Output.Work_Position := TRUE;
		CC1_Output.o_Clamp_WP := FALSE;
		END_IF
	END_IF
	IF (Start_Pb AND CC3_Input.Auto_Sel AND TR_20_Deg AND CC1_Output.Work_Position) THEN
		CC3_Output.o_Clamp_WP := TRUE;
		Cyl_Delay[13](IN:= CC3_Output.o_Clamp_WP, PT:= T#1S, Q=> , ET=> );
		IF Cyl_Delay[13].Q THEN
		CC3_Input.i_Declamp1_Fbk := CC3_Input.i_Declamp2_Fbk := CC3_Input.i_Declamp3_Fbk := CC3_Output.Home_Position := FALSE;
		CC3_Input.i_Clamp1_Fbk := CC3_Input.i_Clamp2_Fbk := CC3_Input.i_Clamp3_Fbk := CC3_Output.Work_Position := TRUE;
		CC3_Output.o_Clamp_WP := FALSE;
		END_IF
	END_IF
	IF (Start_Pb AND CC5_Input.Auto_Sel AND TR_20_Deg AND CC3_Output.Work_Position) THEN
		CC5_Output.o_Clamp_WP := TRUE;
		Cyl_Delay[14](IN:= CC5_Output.o_Clamp_WP, PT:= T#1S, Q=> , ET=> );
		IF Cyl_Delay[14].Q THEN
		CC5_Input.i_Declamp1_Fbk := CC5_Input.i_Declamp2_Fbk := CC5_Input.i_Declamp3_Fbk := CC5_Output.Home_Position := FALSE;
		CC5_Input.i_Clamp1_Fbk := CC5_Input.i_Clamp2_Fbk := CC5_Input.i_Clamp3_Fbk := CC5_Output.Work_Position := TRUE;
		CC5_Output.o_Clamp_WP := FALSE;
		END_IF
	END_IF
	IF (Start_Pb AND CC2_Input.Auto_Sel AND TR_80_Deg AND Part2_Load_Comp AND Roller_Down AND CC5_Output.Work_Position) THEN
		CC2_Output.o_Clamp_WP := TRUE;
		Cyl_Delay[15](IN:= CC2_Output.o_Clamp_WP, PT:= T#1S, Q=> , ET=> );
		IF Cyl_Delay[15].Q THEN
		CC2_Input.i_Declamp1_Fbk := CC2_Input.i_Declamp2_Fbk := CC2_Input.i_Declamp3_Fbk := CC2_Output.Home_Position := FALSE;
		CC2_Input.i_Clamp1_Fbk := CC2_Input.i_Clamp2_Fbk := CC2_Input.i_Clamp3_Fbk := CC2_Output.Work_Position := TRUE;
		CC2_Output.o_Clamp_WP := FALSE;
		END_IF
	END_IF
	IF (Start_Pb AND CC4_Input.Auto_Sel AND TR_80_Deg AND Roller_Down AND CC2_Output.Work_Position) THEN
		CC4_Output.o_Clamp_WP := TRUE;
		Cyl_Delay[16](IN:= CC4_Output.o_Clamp_WP, PT:= T#1S, Q=> , ET=> );
		IF Cyl_Delay[16].Q THEN
		CC4_Input.i_Declamp1_Fbk := CC4_Input.i_Declamp2_Fbk := CC4_Input.i_Declamp3_Fbk := CC4_Output.Home_Position := FALSE;
		CC4_Input.i_Clamp1_Fbk := CC4_Input.i_Clamp2_Fbk := CC4_Input.i_Clamp3_Fbk := CC4_Output.Work_Position := TRUE;
		CC4_Output.o_Clamp_WP := FALSE;
		END_IF
	END_IF
	IF (Start_Pb AND CC6_Input.Auto_Sel AND TR_80_Deg AND Roller_Down AND CC4_Output.Work_Position) THEN
		CC6_Output.o_Clamp_WP := TRUE;
		Cyl_Delay[17](IN:= CC6_Output.o_Clamp_WP, PT:= T#1S, Q=> , ET=> );
		IF Cyl_Delay[17].Q THEN
		CC6_Input.i_Declamp1_Fbk := CC6_Input.i_Declamp2_Fbk := CC6_Input.i_Declamp3_Fbk := CC6_Output.Home_Position := FALSE;
		CC6_Input.i_Clamp1_Fbk := CC6_Input.i_Clamp2_Fbk := CC6_Input.i_Clamp3_Fbk := CC6_Output.Work_Position := TRUE;
		CC6_Output.o_Clamp_WP := FALSE;
		END_IF
	END_IF
	IF (CC5_Input.Auto_Sel AND TT_180_Deg AND TR_0_Deg AND Robot_Weld_Comp) THEN
		CC5_Output.o_Clamp_HP := TRUE;
		Cyl_Delay[18](IN:= CC5_Output.o_Clamp_HP, PT:= T#1S, Q=> , ET=> );
		IF Cyl_Delay[18].Q THEN
		CC5_Input.i_Clamp1_Fbk := CC5_Input.i_Clamp2_Fbk := CC5_Input.i_Clamp3_Fbk := CC5_Output.Work_Position := FALSE;
		CC5_Input.i_Declamp1_Fbk := CC5_Input.i_Declamp2_Fbk := CC5_Input.i_Declamp3_Fbk := CC5_Output.Home_Position := TRUE;
		CC5_Output.o_clamp_HP := FALSE;
		END_IF
	END_IF
	IF (CC3_Input.Auto_Sel AND TT_180_Deg AND TR_0_Deg AND Robot_Weld_Comp) THEN
		CC3_Output.o_Clamp_HP := TRUE;
		Cyl_Delay[19](IN:= CC3_Output.o_Clamp_HP, PT:= T#1S, Q=> , ET=> );
		IF Cyl_Delay[19].Q THEN
		CC3_Input.i_Clamp1_Fbk := CC3_Input.i_Clamp2_Fbk := CC3_Input.i_Clamp3_Fbk := CC3_Output.Work_Position := FALSE;
		CC3_Input.i_Declamp1_Fbk := CC3_Input.i_Declamp2_Fbk := CC3_Input.i_Declamp3_Fbk := CC3_Output.Home_Position := TRUE;
		CC3_Output.o_clamp_HP := FALSE;
		END_IF
	END_IF
	IF (CC1_Input.Auto_Sel AND TT_180_Deg AND TR_0_Deg AND Robot_Weld_Comp) THEN
		CC1_Output.o_Clamp_HP := TRUE;
		Cyl_Delay[20](IN:= CC1_Output.o_Clamp_HP, PT:= T#1S, Q=> , ET=> );
		IF Cyl_Delay[20].Q THEN
		CC1_Input.i_Clamp1_Fbk := CC1_Input.i_Clamp2_Fbk := CC1_Input.i_Clamp3_Fbk := CC1_Output.Work_Position := FALSE;
		CC1_Input.i_Declamp1_Fbk := CC1_Input.i_Declamp2_Fbk := CC1_Input.i_Declamp3_Fbk := CC1_Output.Home_Position := TRUE;
		CC1_Output.o_clamp_HP := FALSE;
		END_IF
	END_IF
	IF (CC1_Output.Home_Position AND CC3_Output.Home_Position AND CC5_Output.Home_Position AND Roller_Up AND Part1_Unload_Comp AND TR_45_Deg AND TT_180_Deg AND Robot_Weld_Comp) THEN
		CC6_Output.o_Clamp_HP := TRUE;
		Cyl_Delay[21](IN:= CC6_Output.o_Clamp_HP, PT:= T#1S, Q=> , ET=> );
		IF Cyl_Delay[21].Q THEN
		CC6_Input.i_Clamp1_Fbk := CC6_Input.i_Clamp2_Fbk := CC6_Input.i_Clamp3_Fbk := CC6_Output.Work_Position := FALSE;
		CC6_Input.i_Declamp1_Fbk := CC6_Input.i_Declamp2_Fbk := CC6_Input.i_Declamp3_Fbk := CC6_Output.Home_Position := TRUE;
		CC6_Output.o_clamp_HP := FALSE;
		END_IF
	END_IF
	IF (CC6_Output.Home_Position AND Roller_Up AND Part1_Unload_Comp AND TR_45_Deg AND TT_180_Deg AND Robot_Weld_Comp) THEN
		CC4_Output.o_Clamp_HP := TRUE;
		Cyl_Delay[22](IN:= CC4_Output.o_Clamp_HP, PT:= T#1S, Q=> , ET=> );
		IF Cyl_Delay[22].Q THEN
		CC4_Input.i_Clamp1_Fbk := CC4_Input.i_Clamp2_Fbk := CC4_Input.i_Clamp3_Fbk := CC4_Output.Work_Position := FALSE;
		CC4_Input.i_Declamp1_Fbk := CC4_Input.i_Declamp2_Fbk := CC4_Input.i_Declamp3_Fbk := CC4_Output.Home_Position := TRUE;
		CC4_Output.o_clamp_HP := FALSE;
		END_IF
	END_IF
	IF (CC4_Output.Home_Position AND Roller_Up AND Part1_Unload_Comp AND TR_45_Deg AND TT_180_Deg AND Robot_Weld_Comp) THEN
		CC2_Output.o_Clamp_HP := TRUE;
		Cyl_Delay[23](IN:= CC2_Output.o_Clamp_HP, PT:= T#1S, Q=> , ET=> );
		IF Cyl_Delay[23].Q THEN
		CC2_Input.i_Clamp1_Fbk := CC2_Input.i_Clamp2_Fbk := CC2_Input.i_Clamp3_Fbk := CC2_Output.Work_Position := FALSE;
		CC2_Input.i_Declamp1_Fbk := CC2_Input.i_Declamp2_Fbk := CC2_Input.i_Declamp3_Fbk := CC2_Output.Home_Position := TRUE;
		CC2_Output.o_clamp_HP := FALSE;
		END_IF
	END_IF

END_CASE

END_FUNCTION_BLOCK

// ---- POUs/TurnTable.TcPOU
FUNCTION_BLOCK TurnTable
VAR_INPUT

	TT_0_Deg  			: BOOL;						//TurnTable at 0 degree
	TT_180_Deg 			: BOOL;						//TurnTable at 180 degree
	Part_Load_Comp 		: BOOL;						//OP710 Part Load Complete
	Part_Unload_Comp 	: BOOL;						//OP710 Part Unload Complete
	Pickup_Comp 		: BOOL;						//Robot Part Pickup Complete
	Roller_Down			: BOOL;						//Roller door Down position
	Roller_Up			: BOOL;						//Roller door Up position
	Fix_Home_Position 	: BOOL;
	Fix_Work_Position 	: BOOL;
	TR_0_Deg  			: BOOL;						//Trunnion at 0 degree
END_VAR

VAR_OUTPUT
	TT_0_Deg_Cmd  : BOOL;						//Trunnion rotate to 0 degree
	TT_180_Deg_Cmd : BOOL;						//Trunnion rotate to 180 degree
END_VAR

VAR
	TT_Rot_Delay : ARRAY [0..5] OF TON;							// TurnTable rotation delay
END_VAR

CASE Fix_Sel OF
	
	0: 

IF (TT_0_Deg AND TR_0_Deg AND Part_Load_Comp AND Fix_Work_Position AND Roller_Down AND Start_Pb) THEN
	TT_180_Deg_Cmd := TRUE;
	TT_Rot_Delay[0](IN:= TT_180_Deg_Cmd , PT:= T#1S, Q=> , ET=> );
	IF TT_Rot_Delay[0].Q THEN
	TT_0_Deg := FALSE;
	TT_180_Deg := TRUE;
	TT_180_Deg_Cmd := FALSE;
	END_IF	
ELSIF (TT_180_Deg AND Pickup_Comp AND Roller_Up AND Fix_Home_Position) THEN
	TT_0_Deg_Cmd := TRUE;
	TT_Rot_Delay[1](IN:= TT_0_Deg_Cmd , PT:= T#1S, Q=> , ET=> );
	IF TT_Rot_Delay[1].Q THEN
	TT_180_Deg := FALSE;
	TT_0_Deg := TRUE;
	TT_0_Deg_Cmd := FALSE;
	END_IF
END_IF
	Fix_Sel := 0;

	1: 

IF (TT_180_Deg AND TR_0_Deg AND Part_Load_Comp AND Fix_Work_Position AND Roller_Down AND Start_Pb) THEN
	TT_180_Deg_Cmd := TRUE;
	TT_Rot_Delay[2](IN:= TT_180_Deg_Cmd , PT:= T#1S, Q=> , ET=> );
	IF TT_Rot_Delay[2].Q THEN
	TT_0_Deg := FALSE;
	TT_180_Deg := TRUE;
	TT_180_Deg_Cmd := FALSE;
	END_IF	
ELSIF (TT_0_Deg AND Pickup_Comp AND Roller_Up AND Fix_Home_Position) THEN
	TT_180_Deg_Cmd := TRUE;
	TT_Rot_Delay[3](IN:= TT_180_Deg_Cmd , PT:= T#1S, Q=> , ET=> );
	IF TT_Rot_Delay[3].Q THEN
	TT_0_Deg := FALSE;
	TT_180_Deg := TRUE;
	TT_180_Deg_Cmd := FALSE;
	END_IF
END_IF
	Fix_Sel := 1;

END_CASE

END_FUNCTION_BLOCK

// ---- POUs/Trunnion.TcPOU
FUNCTION_BLOCK Trunnion
VAR_INPUT
	TR_0_Deg  				: BOOL;						//Trunnion at 0 degree
	TR_20_Deg 				: BOOL;						//Trunnion at -20 degree
	TR_45_Deg 				: BOOL;						//Trunnion at 45 degree
	TR_50_Deg 				: BOOL;						//Trunnion at 50 degree
	TR_80_Deg 				: BOOL;						//Trunnion at 80 degree
	Load_Comp1 				: BOOL;						//Fixture Part-1 Load Complete
	Load_Comp2 				: BOOL;						//Fixture Part-2 Load Complete
	Unload_Comp1 			: BOOL;						//Fixture Part-1 Unload Complete
	Unload_Comp2 			: BOOL;						//Fixture Part-2 Unload Complete
	Roller_Up 				: BOOL;						//Roller Door Up position
	Roller_Down 			: BOOL;						//Roller Door Down position
	Weld_Comp 				: BOOL;						//Robot Weld Complete
	Pickup_Comp1 			: BOOL;						//Robot Pickup Complete-1
	Pickup_Comp2 			: BOOL;						//Robot Pickup Complete-2
END_VAR

VAR_OUTPUT
	TR_0_Deg_Cmd  			: BOOL;						//Trunnion rotate to 0 degree
	TR_20_Deg_Cmd 			: BOOL;						//Trunnion rotate to -20 degree
	TR_45_Deg_Cmd 			: BOOL;						//Trunnion rotate to 45 degree
	TR_50_Deg_Cmd 			: BOOL;						//Trunnion rotate to 50 degree
	TR_80_Deg_Cmd 			: BOOL;						//Trunnion rotate to 80 degree
END_VAR

VAR
	TR_Rot_Delay : ARRAY [0..10] OF TON;							// Trunnion rotation delay
	
END_VAR

CASE Fix_Sel OF
	
	0: 
IF (TR_0_Deg AND (NOT Load_Comp1) AND (NOT Weld_Comp) AND Start_Pb) THEN
	TR_20_Deg_Cmd := TRUE;
	TR_Rot_Delay[0](IN:= TR_20_Deg_Cmd, PT:= T#1S , Q=> , ET=> );
	IF TR_Rot_Delay[0].Q THEN
	TR_0_Deg := FALSE;
	TR_20_Deg_Cmd := FALSE;
	TR_20_Deg := TRUE;
	END_IF
ELSIF (TR_20_Deg AND Load_Comp1 AND Start_Pb) THEN
	TR_80_Deg_Cmd := TRUE;
	TR_Rot_Delay[1](IN:= TR_80_Deg_Cmd, PT:= T#1S, Q=> , ET=> );
	IF TR_Rot_Delay[1].Q THEN
	TR_20_Deg := FALSE;
	TR_80_Deg_Cmd := FALSE;
	TR_80_Deg := TRUE;
	END_IF
ELSIF (TR_80_Deg AND Load_Comp2 AND Roller_Down AND Start_Pb) THEN
	TR_0_Deg_Cmd := TRUE;
	TR_Rot_Delay[2](IN:= TR_0_Deg_Cmd, PT:= T#1S, Q=> , ET=> );
	IF TR_Rot_Delay[2].Q THEN
	TR_80_Deg := FALSE;
	TR_0_Deg_Cmd := FALSE;
	TR_0_Deg := TRUE;
	END_IF
ELSIF (TR_0_Deg AND Roller_Up AND Unload_Comp1 AND Weld_Comp AND Pickup_Comp1 AND NOT Pickup_Comp2) THEN
	TR_45_Deg_Cmd := TRUE;
	TR_Rot_Delay[3](IN:= TR_45_Deg_Cmd, PT:= T#1S, Q=> , ET=> );
	IF TR_Rot_Delay[3].Q THEN
	TR_0_Deg := FALSE;
	TR_45_Deg_Cmd := FALSE;
	TR_45_Deg := TRUE;
	END_IF
ELSIF (TR_45_Deg AND Roller_Up AND Pickup_Comp2) THEN
	TR_0_Deg_Cmd := TRUE;
	TR_Rot_Delay[4](IN:= TR_0_Deg_Cmd, PT:= T#1S, Q=> , ET=> );
	IF TR_Rot_Delay[4].Q THEN
	TR_45_Deg := FALSE;
	TR_0_Deg_Cmd := FALSE;
	TR_0_Deg := TRUE;
	END_IF
END_IF
	Fix_Sel := 0;
	
	
	1: 
IF (TR_0_Deg AND (NOT Load_Comp1) AND (NOT Weld_Comp) AND Start_Pb) THEN
	TR_20_Deg_Cmd := TRUE;
	TR_Rot_Delay[5](IN:= TR_20_Deg_Cmd, PT:= T#1S, Q=> , ET=> );
	IF TR_Rot_Delay[5].Q THEN
	TR_0_Deg := FALSE;
	TR_20_Deg_Cmd := FALSE;
	TR_20_Deg := TRUE;
	END_IF
ELSIF (TR_20_Deg AND Load_Comp1 AND Start_Pb) THEN
	TR_50_Deg_Cmd := TRUE;
	TR_Rot_Delay[6](IN:= TR_50_Deg_Cmd, PT:= T#1S, Q=> , ET=> );
	IF TR_Rot_Delay[6].Q THEN
	TR_20_Deg := FALSE;
	TR_50_Deg_Cmd := FALSE;
	TR_50_Deg := TRUE;
	END_IF
ELSIF (TR_50_Deg AND Load_Comp2 AND Roller_Down AND Start_Pb) THEN
	TR_0_Deg_Cmd := TRUE;
	TR_Rot_Delay[7](IN:= TR_0_Deg_Cmd, PT:= T#1S, Q=> , ET=> );
	IF TR_Rot_Delay[7].Q THEN
	TR_50_Deg := FALSE;
	TR_0_Deg_Cmd := FALSE;
	TR_0_Deg := TRUE;
	END_IF
ELSIF (TR_0_Deg AND Roller_Up AND Unload_Comp1 AND Weld_Comp AND Pickup_Comp1 AND NOT Pickup_Comp2) THEN
	TR_50_Deg_Cmd := TRUE;
	TR_Rot_Delay[8](IN:= TR_50_Deg_Cmd, PT:= T#1S, Q=> , ET=> );
	IF TR_Rot_Delay[8].Q THEN
	TR_0_Deg := FALSE;
	TR_50_Deg_Cmd := FALSE;
	TR_50_Deg := TRUE;
	END_IF
ELSIF (TR_50_Deg AND Roller_Up AND Pickup_Comp2) THEN
	TR_0_Deg_Cmd := TRUE;
	TR_Rot_Delay[9](IN:= TR_0_Deg_Cmd, PT:= T#1S, Q=> , ET=> );
	IF TR_Rot_Delay[9].Q THEN
	TR_50_Deg := FALSE;
	TR_0_Deg_Cmd := FALSE;
	TR_0_Deg := TRUE;
	END_IF
END_IF
	Fix_Sel := 1;
END_CASE

END_FUNCTION_BLOCK

// ---- POUs/RollerDoor.TcPOU
FUNCTION_BLOCK RollerDoor
VAR_INPUT

	Roller_Up  			: BOOL;						//Roller Door Up position
	Roller_Down 		: BOOL;						//Roller Door Down position
	Part_Load_Comp 		: BOOL;						//OP710 Part Load Complete
	Part_Unload_Comp 	: BOOL;						//OP710 Part Unload Complete
	Weld_Comp 			: BOOL;						//Robot Weld Complete
	TR_0_Deg  			: BOOL;						//Trunnion at 0 degree
	TR_50_Deg  			: BOOL;						//Trunnion at 50 degree
	TR_80_Deg  			: BOOL;						//Trunnion at 80 degree
	TT_0_Deg  			: BOOL;						//TurnTable at 0 degree
	TT_180_Deg  		: BOOL;						//TurnTable at 180 degree
	
END_VAR

VAR_OUTPUT
	Roller_Up_Cmd  : BOOL;						//Roller Door Up Command
	Roller_Down_Cmd : BOOL;						//Roller Door Down Command
END_VAR

VAR
	Roller_Delay : ARRAY [0..5] OF TON;						// Roller Door Up/Down delay
END_VAR

CASE Fix_Sel OF
	
	0: 
IF (Roller_Up AND Part_Load_Comp AND TR_80_Deg AND TT_0_Deg AND Start_Pb) THEN
	Roller_Down_Cmd := TRUE;
	Roller_Delay[0](IN:= Roller_Down_Cmd , PT:= T#1S, Q=> , ET=> );
	IF Roller_Delay[0].Q THEN
	Roller_Up := FALSE;
	Roller_Down := TRUE;
	Roller_Down_Cmd := FALSE;
	END_IF	
ELSIF (Roller_Down AND Weld_Comp AND TR_0_Deg AND TT_180_Deg AND Start_Pb) THEN
	Roller_Up_Cmd := TRUE;
	Roller_Delay[1](IN:= Roller_Up_Cmd , PT:= T#1S, Q=> , ET=> );
	IF Roller_Delay[1].Q THEN
	Roller_Down := FALSE;
	Roller_Up := TRUE;
	Roller_Up_Cmd := FALSE;
	END_IF
END_IF
	Fix_Sel := 0;

	1:
IF (Roller_Up AND Part_Load_Comp AND TR_50_Deg AND TT_180_Deg AND Start_Pb) THEN
	Roller_Down_Cmd := TRUE;
	Roller_Delay[2](IN:= Roller_Down_Cmd , PT:= T#1S, Q=> , ET=> );
	IF Roller_Delay[2].Q THEN
	Roller_Up := FALSE;
	Roller_Down := TRUE;
	Roller_Down_Cmd := FALSE;
	END_IF	
ELSIF (Roller_Down AND Weld_Comp AND TR_0_Deg AND TT_0_Deg AND Start_Pb) THEN
	Roller_Up_Cmd := TRUE;
	Roller_Delay[3](IN:= Roller_Up_Cmd , PT:= T#1S, Q=> , ET=> );
	IF Roller_Delay[3].Q THEN
	Roller_Down := FALSE;
	Roller_Up := TRUE;
	Roller_Up_Cmd := FALSE;
	END_IF
END_IF
	Fix_Sel := 1;
END_CASE

END_FUNCTION_BLOCK

// ---- POUs/Robot_Weld.TcPOU
FUNCTION_BLOCK Robot_Weld

VAR_INPUT
	Robot_1_In			:	Weld_Robot;
	Part_Unload_Comp	:	BOOL;
END_VAR

VAR_OUTPUT
	Robot_1_Out			:	Weld_Robot;	
END_VAR

VAR
	Weld_Delay			:	TON;
END_VAR

CASE Robot_1_In.i_Prg_No OF
	101:
		IF (Robot_1_In.i_Area_Ok AND Robot_1_In.i_Start) THEN
		Robot_1_In.i_Home := FALSE;
		Weld_Delay(IN:= Robot_1_In.i_Start, PT:= T#1S, Q=> , ET=> );
		IF Weld_Delay.Q THEN
		Robot_1_Out.o_Weld_Comp := TRUE;
		Robot_1_In.i_Home := TRUE;
		END_IF
		END_IF
		IF (Robot_1_In.i_Home AND Part_Unload_Comp) THEN
		Robot_1_Out.o_Weld_Comp := FALSE;	
		END_IF
		Robot_1_In.i_Prg_No := 101;
	102:
		IF (Robot_1_In.i_Area_Ok AND Robot_1_In.i_Start) THEN
		Robot_1_In.i_Home := FALSE;
		Weld_Delay(IN:= Robot_1_In.i_Start, PT:= T#1S, Q=> , ET=> );
		IF Weld_Delay.Q THEN
		Robot_1_Out.o_Weld_Comp := TRUE;
		Robot_1_In.i_Home := TRUE;
		END_IF
		END_IF
		IF (Robot_1_In.i_Home AND Part_Unload_Comp) THEN
		Robot_1_Out.o_Weld_Comp := FALSE;	
		END_IF
		Robot_1_In.i_Prg_No := 102;
END_CASE

END_FUNCTION_BLOCK

// ---- POUs/Robot_MH.TcPOU
FUNCTION_BLOCK Robot_MH

VAR_INPUT
	Robot_1_In			: MH_Robot;
	Part_Unload_Comp	: BOOL;
END_VAR

VAR_OUTPUT
	Robot_1_Out			: MH_Robot;	
END_VAR

VAR
	Pickup_Delay			: ARRAY [0..5] OF TON;
END_VAR

CASE Robot_1_In.i_Prg_No OF
	101:
		IF (Robot_1_In.i_Home AND Robot_1_In.i_Area_Ok1 AND Robot_1_In.i_Start) THEN
		Pickup_Delay[0](IN:= Robot_1_In.i_Start, PT:= T#1S, Q=> , ET=> );
		IF Pickup_Delay[0].Q THEN
		Robot_1_In.i_Home := FALSE;
		Robot_1_Out.o_Pickup_Comp1 := TRUE;
		Robot_1_In.i_Home := TRUE;
		END_IF
		END_IF
		IF (Robot_1_In.i_Home AND Robot_1_In.i_Area_Ok2 AND Robot_1_In.i_Start) THEN
		Pickup_Delay[1](IN:= Robot_1_In.i_Start, PT:= T#1S, Q=> , ET=> );
		IF Pickup_Delay[1].Q THEN
		Robot_1_In.i_Home := FALSE;
		Robot_1_Out.o_Pickup_Comp2 := TRUE;
		Robot_1_In.i_Home := TRUE;
		END_IF
		END_IF
		IF (Robot_1_In.i_Home AND Part_Unload_Comp) THEN
		Robot_1_Out.o_Pickup_Comp1 := FALSE;
		Robot_1_Out.o_Pickup_Comp2 := FALSE;	
		END_IF
	102:
		IF (Robot_1_In.i_Home AND Robot_1_In.i_Area_Ok1 AND Robot_1_In.i_Start) THEN
		Pickup_Delay[2](IN:= Robot_1_In.i_Start, PT:= T#1S, Q=> , ET=> );
		IF Pickup_Delay[2].Q THEN
		Robot_1_In.i_Home := FALSE;
		Robot_1_Out.o_Pickup_Comp1 := TRUE;
		Robot_1_In.i_Home := TRUE;
		END_IF
		END_IF
		IF (Robot_1_In.i_Home AND Robot_1_In.i_Area_Ok2 AND Robot_1_In.i_Start) THEN
		Pickup_Delay[3](IN:= Robot_1_In.i_Start, PT:= T#1S, Q=> , ET=> );
		IF Pickup_Delay[3].Q THEN
		Robot_1_In.i_Home := FALSE;
		Robot_1_Out.o_Pickup_Comp2 := TRUE;
		Robot_1_In.i_Home := TRUE;
		END_IF
		END_IF
		IF (Robot_1_In.i_Home AND Part_Unload_Comp) THEN
		Robot_1_Out.o_Pickup_Comp1 := FALSE;
		Robot_1_Out.o_Pickup_Comp2 := FALSE;	
		END_IF
END_CASE

END_FUNCTION_BLOCK

// ---- POUs/Auto_Cycle_Fix2.TcPOU
PROGRAM Auto_Cycle_Fix2
VAR
	Fixture_2 : Fix2_FB;
	TurnTable_1: TurnTable;
	Trunnion_1: Trunnion;
	RollerDoor_1: RollerDoor;
	Robot_Weld_1: Robot_Weld;
	Robot_MH_1: Robot_MH;
END_VAR
VAR // added by the converter: edge detectors and wires of the graphical bodies
    _w1, _w2 : BOOL;
END_VAR

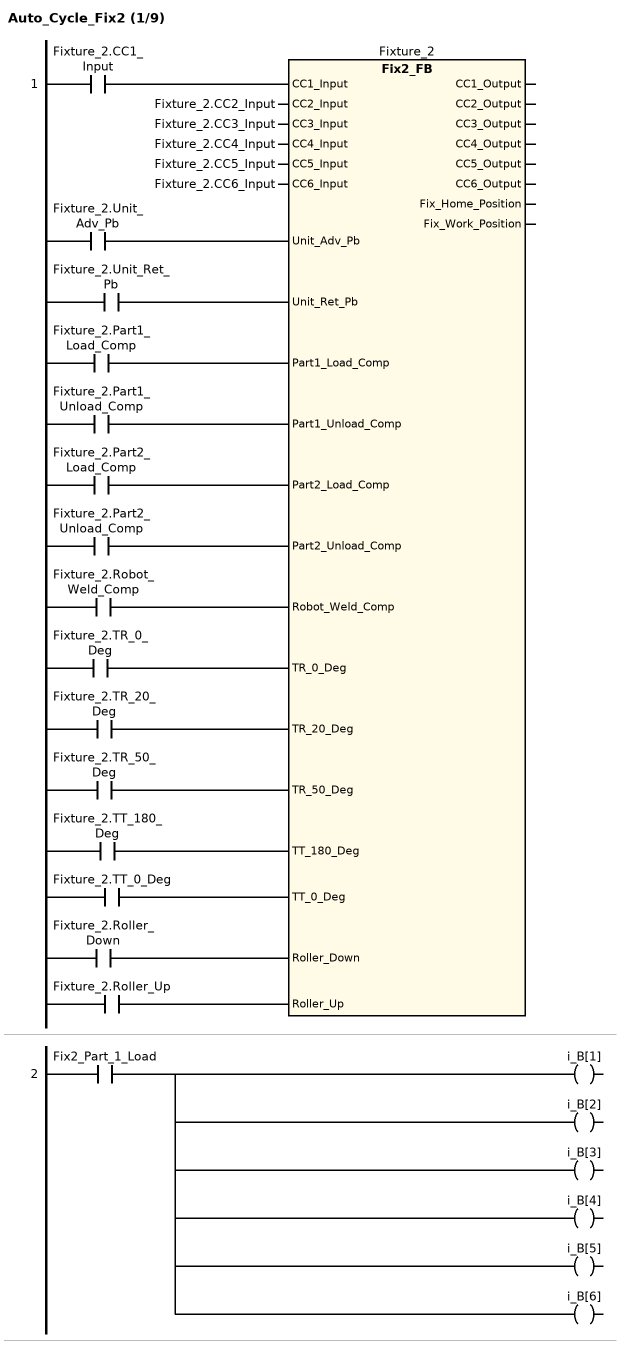
// NETWORK 1
Fixture_2(
    CC1_Input := Fixture_2.CC1_Input,
    CC2_Input := Fixture_2.CC2_Input,
    CC3_Input := Fixture_2.CC3_Input,
    CC4_Input := Fixture_2.CC4_Input,
    CC5_Input := Fixture_2.CC5_Input,
    CC6_Input := Fixture_2.CC6_Input,
    Unit_Adv_Pb := Fixture_2.Unit_Adv_Pb,
    Unit_Ret_Pb := Fixture_2.Unit_Ret_Pb,
    Part1_Load_Comp := Fixture_2.Part1_Load_Comp,
    Part1_Unload_Comp := Fixture_2.Part1_Unload_Comp,
    Part2_Load_Comp := Fixture_2.Part2_Load_Comp,
    Part2_Unload_Comp := Fixture_2.Part2_Unload_Comp,
    Robot_Weld_Comp := Fixture_2.Robot_Weld_Comp,
    TR_0_Deg := Fixture_2.TR_0_Deg,
    TR_20_Deg := Fixture_2.TR_20_Deg,
    TR_50_Deg := Fixture_2.TR_50_Deg,
    TT_180_Deg := Fixture_2.TT_180_Deg,
    TT_0_Deg := Fixture_2.TT_0_Deg,
    Roller_Down := Fixture_2.Roller_Down,
    Roller_Up := Fixture_2.Roller_Up); // Fix2_FB

// NETWORK 2
i_B[1] := Fix2_Part_1_Load;
i_B[2] := Fix2_Part_1_Load;
i_B[3] := Fix2_Part_1_Load;
i_B[4] := Fix2_Part_1_Load;
i_B[5] := Fix2_Part_1_Load;
i_B[6] := Fix2_Part_1_Load;

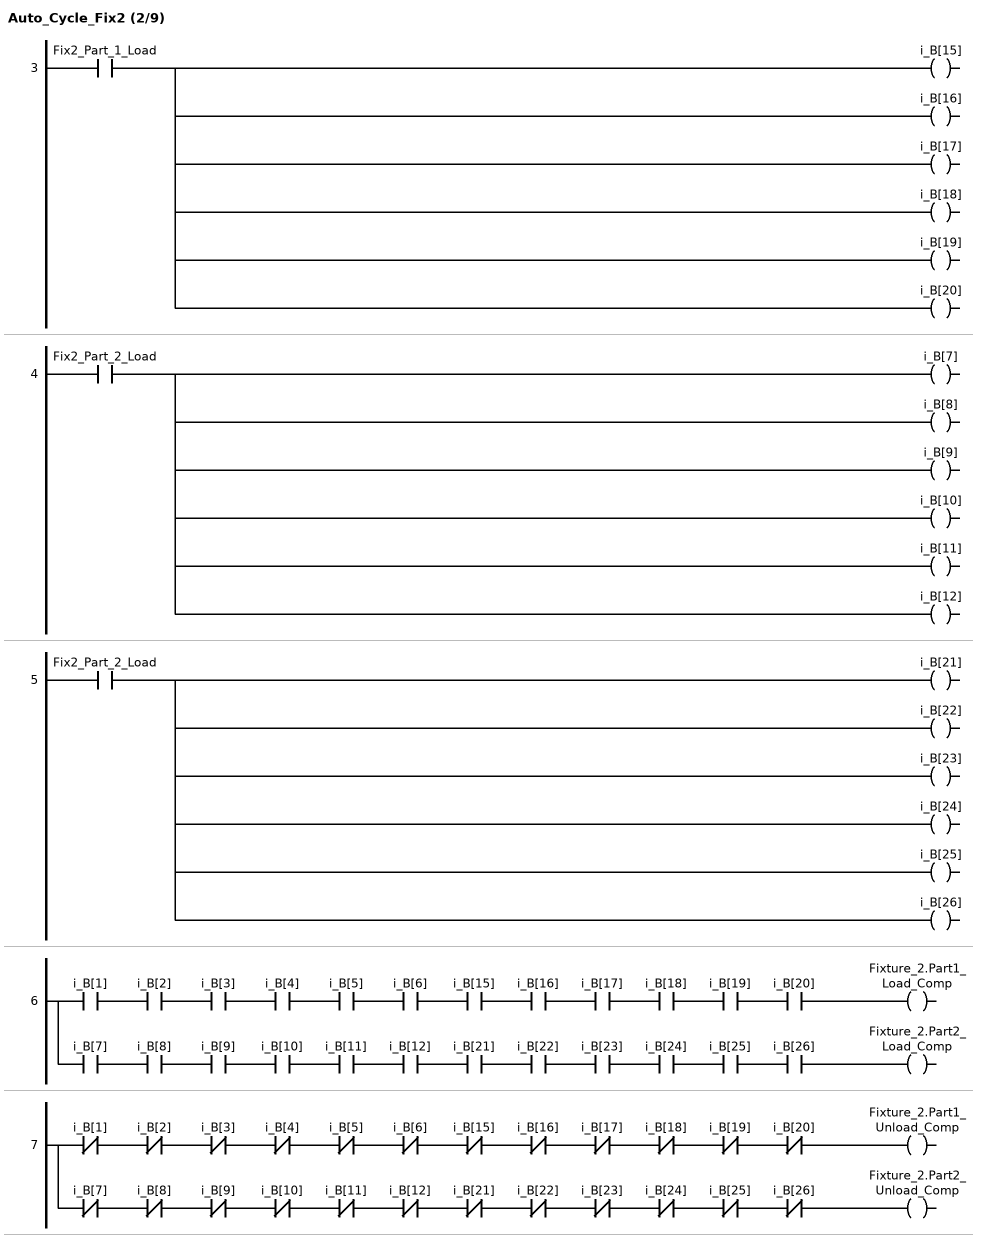
// NETWORK 3
i_B[15] := Fix2_Part_1_Load;
i_B[16] := Fix2_Part_1_Load;
i_B[17] := Fix2_Part_1_Load;
i_B[18] := Fix2_Part_1_Load;
i_B[19] := Fix2_Part_1_Load;
i_B[20] := Fix2_Part_1_Load;

// NETWORK 4
i_B[7] := Fix2_Part_2_Load;
i_B[8] := Fix2_Part_2_Load;
i_B[9] := Fix2_Part_2_Load;
i_B[10] := Fix2_Part_2_Load;
i_B[11] := Fix2_Part_2_Load;
i_B[12] := Fix2_Part_2_Load;

// NETWORK 5
i_B[21] := Fix2_Part_2_Load;
i_B[22] := Fix2_Part_2_Load;
i_B[23] := Fix2_Part_2_Load;
i_B[24] := Fix2_Part_2_Load;
i_B[25] := Fix2_Part_2_Load;
i_B[26] := Fix2_Part_2_Load;

// NETWORK 6
Fixture_2.Part1_Load_Comp := i_B[1] AND i_B[2] AND i_B[3] AND i_B[4] AND i_B[5] AND i_B[6] AND i_B[15] AND i_B[16] AND i_B[17] AND i_B[18] AND i_B[19] AND i_B[20];
Fixture_2.Part2_Load_Comp := i_B[7] AND i_B[8] AND i_B[9] AND i_B[10] AND i_B[11] AND i_B[12] AND i_B[21] AND i_B[22] AND i_B[23] AND i_B[24] AND i_B[25] AND i_B[26];

// NETWORK 7
Fixture_2.Part1_Unload_Comp := NOT i_B[1] AND NOT i_B[2] AND NOT i_B[3] AND NOT i_B[4] AND NOT i_B[5] AND NOT i_B[6] AND NOT i_B[15] AND NOT i_B[16] AND NOT i_B[17] AND NOT i_B[18] AND NOT i_B[19] AND NOT i_B[20];
Fixture_2.Part2_Unload_Comp := NOT i_B[7] AND NOT i_B[8] AND NOT i_B[9] AND NOT i_B[10] AND NOT i_B[11] AND NOT i_B[12] AND NOT i_B[21] AND NOT i_B[22] AND NOT i_B[23] AND NOT i_B[24] AND NOT i_B[25] AND NOT i_B[26];

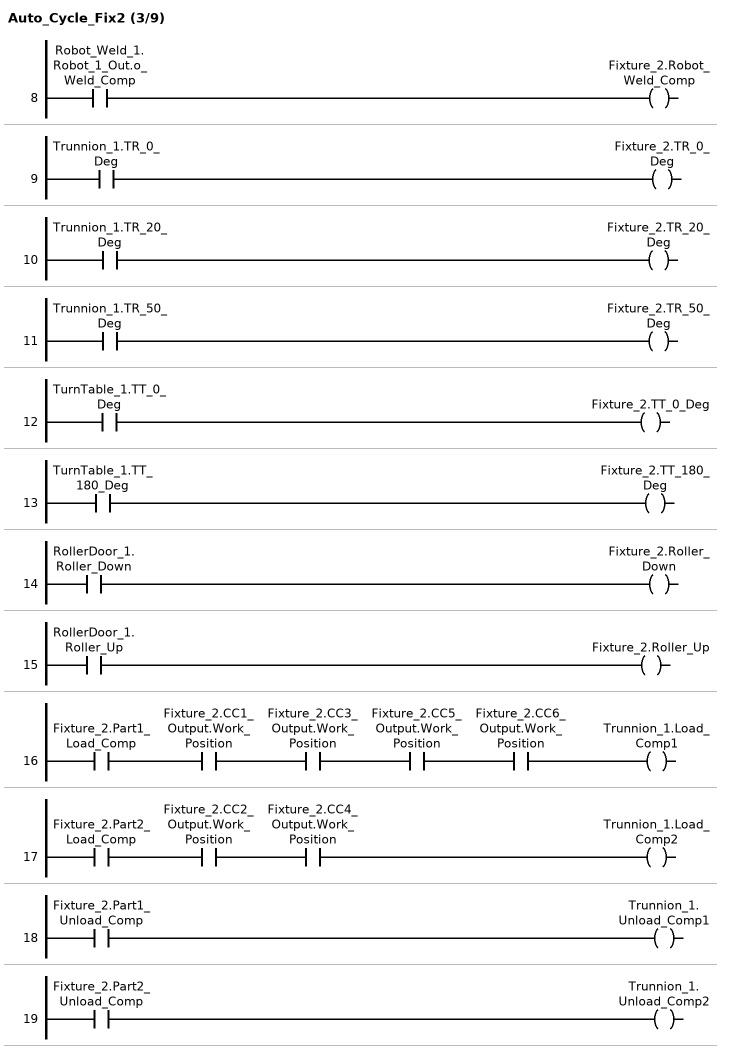
// NETWORK 8
Fixture_2.Robot_Weld_Comp := Robot_Weld_1.Robot_1_Out.o_Weld_Comp;

// NETWORK 9
Fixture_2.TR_0_Deg := Trunnion_1.TR_0_Deg;

// NETWORK 10
Fixture_2.TR_20_Deg := Trunnion_1.TR_20_Deg;

// NETWORK 11
Fixture_2.TR_50_Deg := Trunnion_1.TR_50_Deg;

// NETWORK 12
Fixture_2.TT_0_Deg := TurnTable_1.TT_0_Deg;

// NETWORK 13
Fixture_2.TT_180_Deg := TurnTable_1.TT_180_Deg;

// NETWORK 14
Fixture_2.Roller_Down := RollerDoor_1.Roller_Down;

// NETWORK 15
Fixture_2.Roller_Up := RollerDoor_1.Roller_Up;

// NETWORK 16
Trunnion_1.Load_Comp1 := Fixture_2.Part1_Load_Comp AND Fixture_2.CC1_Output.Work_Position AND Fixture_2.CC3_Output.Work_Position AND Fixture_2.CC5_Output.Work_Position AND Fixture_2.CC6_Output.Work_Position;

// NETWORK 17
Trunnion_1.Load_Comp2 := Fixture_2.Part2_Load_Comp AND Fixture_2.CC2_Output.Work_Position AND Fixture_2.CC4_Output.Work_Position;

// NETWORK 18
Trunnion_1.Unload_Comp1 := Fixture_2.Part1_Unload_Comp;

// NETWORK 19
Trunnion_1.Unload_Comp2 := Fixture_2.Part2_Unload_Comp;

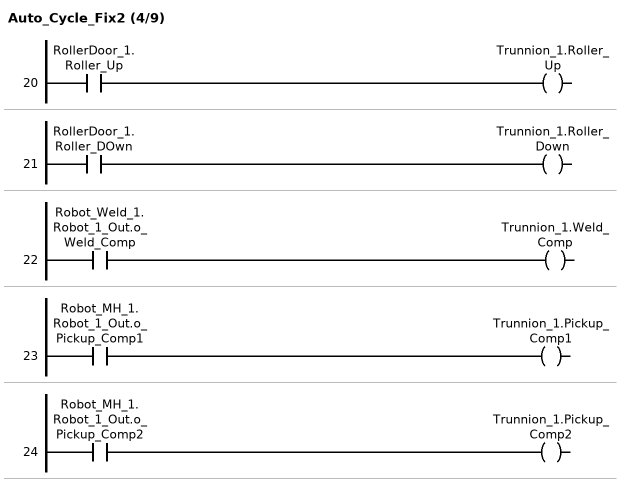
// NETWORK 20
Trunnion_1.Roller_Up := RollerDoor_1.Roller_Up;

// NETWORK 21
Trunnion_1.Roller_Down := RollerDoor_1.Roller_DOwn;

// NETWORK 22
Trunnion_1.Weld_Comp := Robot_Weld_1.Robot_1_Out.o_Weld_Comp;

// NETWORK 23
Trunnion_1.Pickup_Comp1 := Robot_MH_1.Robot_1_Out.o_Pickup_Comp1;

// NETWORK 24
Trunnion_1.Pickup_Comp2 := Robot_MH_1.Robot_1_Out.o_Pickup_Comp2;

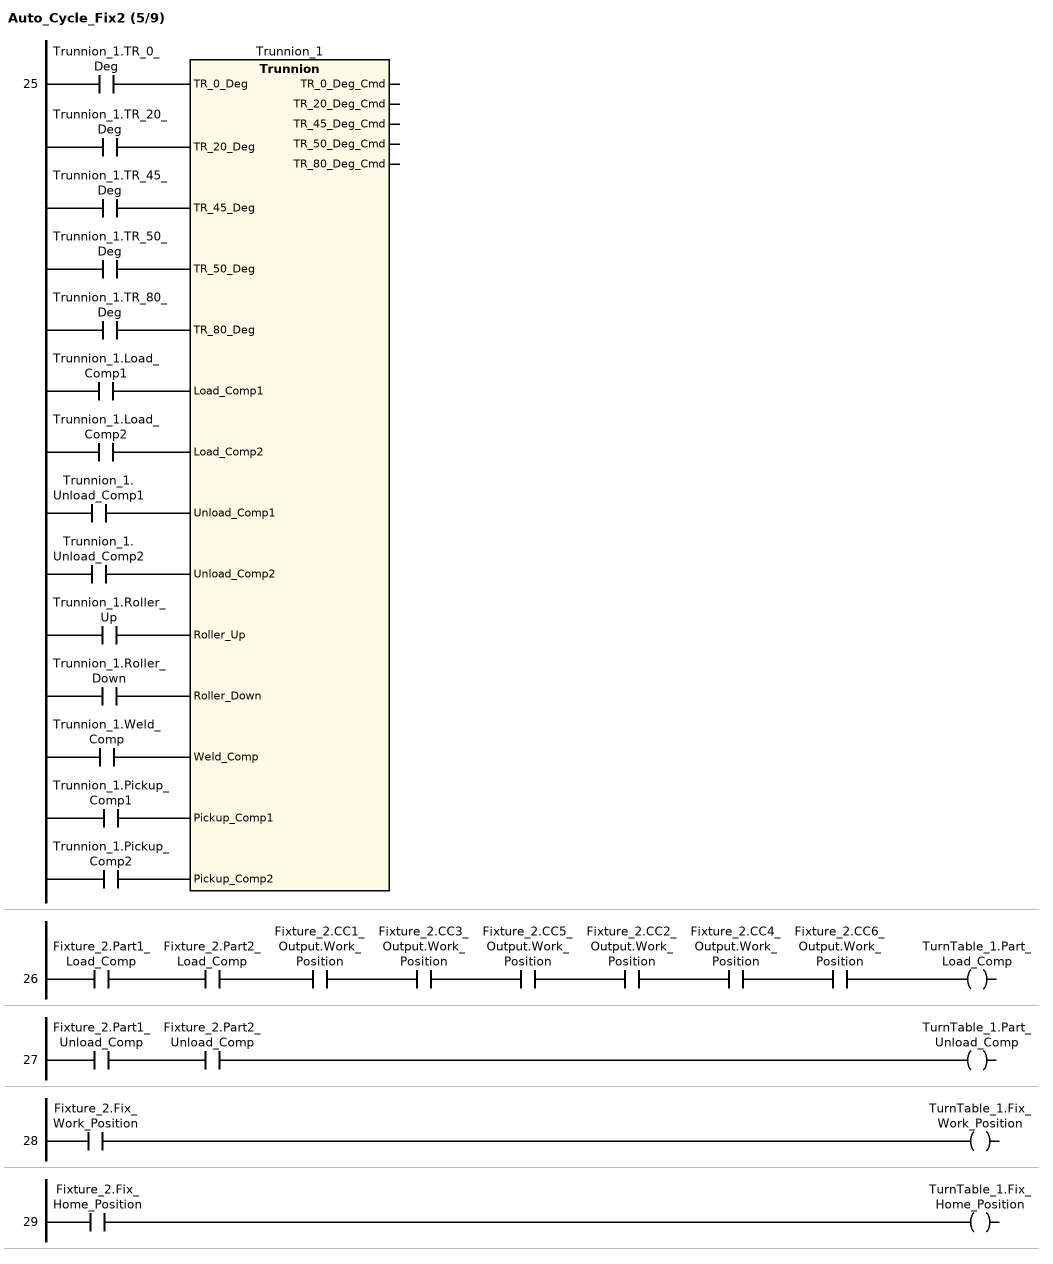
// NETWORK 25
Trunnion_1(
    TR_0_Deg := Trunnion_1.TR_0_Deg,
    TR_20_Deg := Trunnion_1.TR_20_Deg,
    TR_45_Deg := Trunnion_1.TR_45_Deg,
    TR_50_Deg := Trunnion_1.TR_50_Deg,
    TR_80_Deg := Trunnion_1.TR_80_Deg,
    Load_Comp1 := Trunnion_1.Load_Comp1,
    Load_Comp2 := Trunnion_1.Load_Comp2,
    Unload_Comp1 := Trunnion_1.Unload_Comp1,
    Unload_Comp2 := Trunnion_1.Unload_Comp2,
    Roller_Up := Trunnion_1.Roller_Up,
    Roller_Down := Trunnion_1.Roller_Down,
    Weld_Comp := Trunnion_1.Weld_Comp,
    Pickup_Comp1 := Trunnion_1.Pickup_Comp1,
    Pickup_Comp2 := Trunnion_1.Pickup_Comp2); // Trunnion

// NETWORK 26
TurnTable_1.Part_Load_Comp := Fixture_2.Part1_Load_Comp AND Fixture_2.Part2_Load_Comp AND Fixture_2.CC1_Output.Work_Position AND Fixture_2.CC3_Output.Work_Position AND Fixture_2.CC5_Output.Work_Position AND Fixture_2.CC2_Output.Work_Position AND Fixture_2.CC4_Output.Work_Position AND Fixture_2.CC6_Output.Work_Position;

// NETWORK 27
TurnTable_1.Part_Unload_Comp := Fixture_2.Part1_Unload_Comp AND Fixture_2.Part2_Unload_Comp;

// NETWORK 28
TurnTable_1.Fix_Work_Position := Fixture_2.Fix_Work_Position;

// NETWORK 29
TurnTable_1.Fix_Home_Position := Fixture_2.Fix_Home_Position;

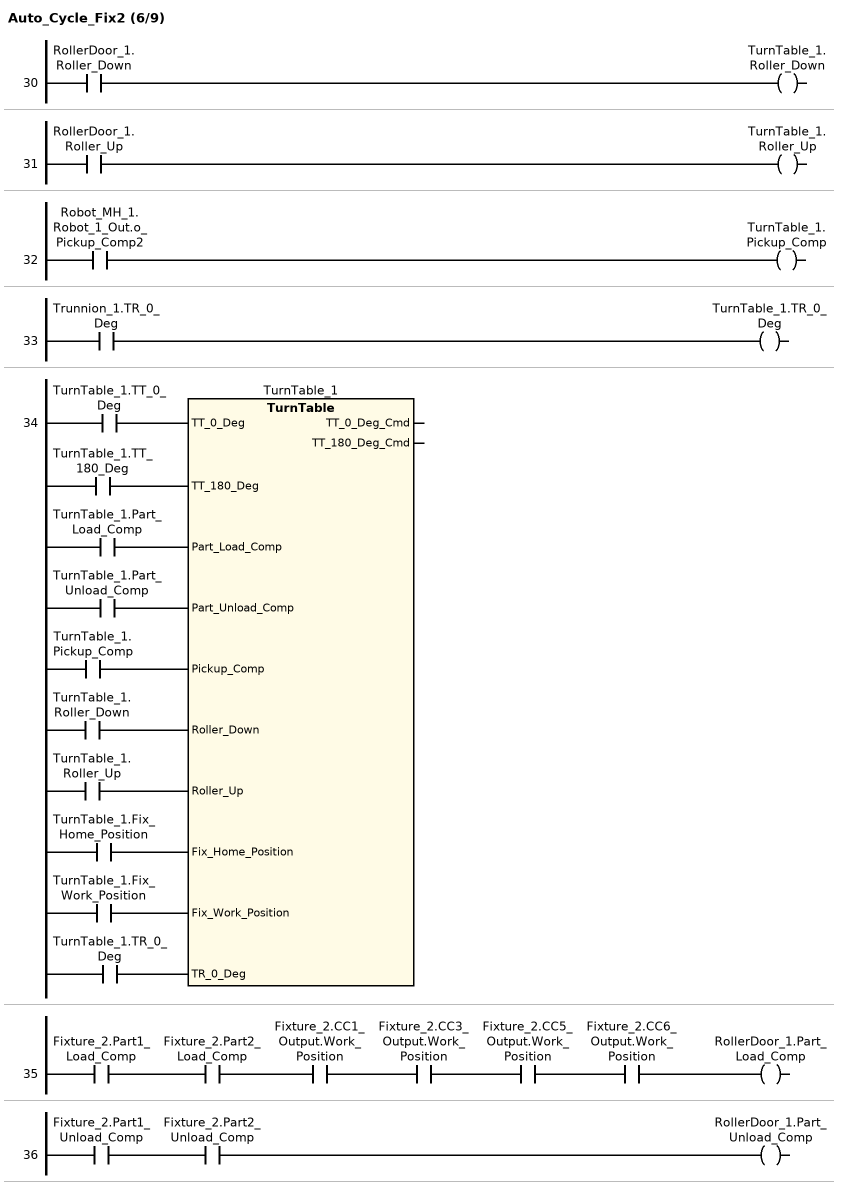
// NETWORK 30
TurnTable_1.Roller_Down := RollerDoor_1.Roller_Down;

// NETWORK 31
TurnTable_1.Roller_Up := RollerDoor_1.Roller_Up;

// NETWORK 32
TurnTable_1.Pickup_Comp := Robot_MH_1.Robot_1_Out.o_Pickup_Comp2;

// NETWORK 33
TurnTable_1.TR_0_Deg := Trunnion_1.TR_0_Deg;

// NETWORK 34
TurnTable_1(
    TT_0_Deg := TurnTable_1.TT_0_Deg,
    TT_180_Deg := TurnTable_1.TT_180_Deg,
    Part_Load_Comp := TurnTable_1.Part_Load_Comp,
    Part_Unload_Comp := TurnTable_1.Part_Unload_Comp,
    Pickup_Comp := TurnTable_1.Pickup_Comp,
    Roller_Down := TurnTable_1.Roller_Down,
    Roller_Up := TurnTable_1.Roller_Up,
    Fix_Home_Position := TurnTable_1.Fix_Home_Position,
    Fix_Work_Position := TurnTable_1.Fix_Work_Position,
    TR_0_Deg := TurnTable_1.TR_0_Deg); // TurnTable

// NETWORK 35
RollerDoor_1.Part_Load_Comp := Fixture_2.Part1_Load_Comp AND Fixture_2.Part2_Load_Comp AND Fixture_2.CC1_Output.Work_Position AND Fixture_2.CC3_Output.Work_Position AND Fixture_2.CC5_Output.Work_Position AND Fixture_2.CC6_Output.Work_Position;

// NETWORK 36
RollerDoor_1.Part_Unload_Comp := Fixture_2.Part1_Unload_Comp AND Fixture_2.Part2_Unload_Comp;

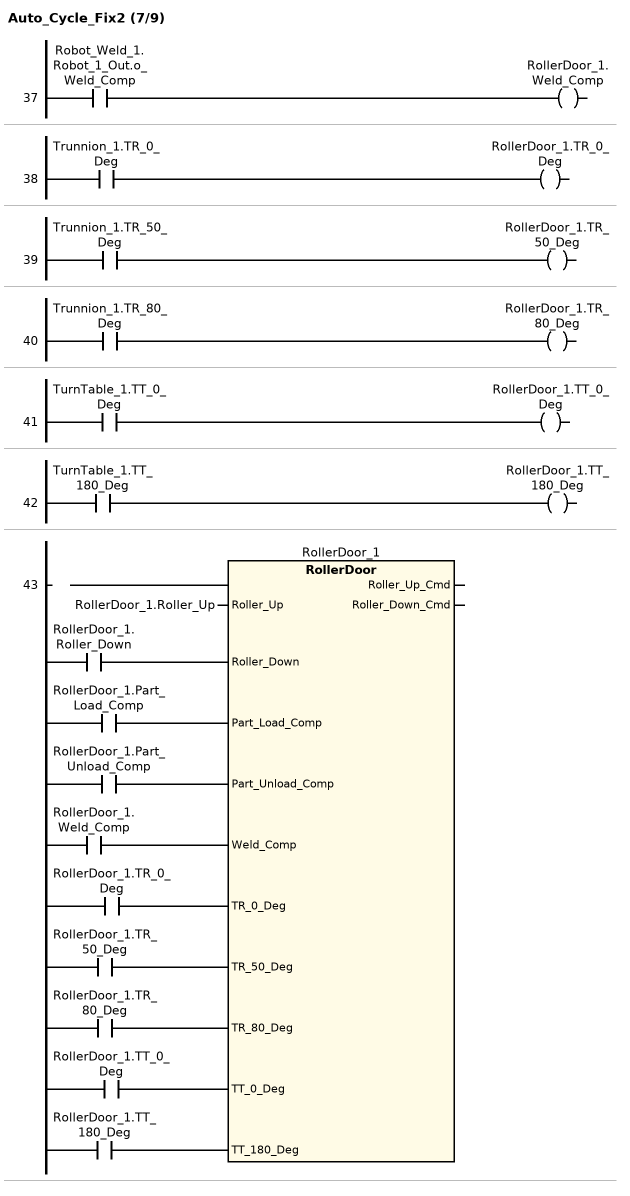
// NETWORK 37
RollerDoor_1.Weld_Comp := Robot_Weld_1.Robot_1_Out.o_Weld_Comp;

// NETWORK 38
RollerDoor_1.TR_0_Deg := Trunnion_1.TR_0_Deg;

// NETWORK 39
RollerDoor_1.TR_50_Deg := Trunnion_1.TR_50_Deg;

// NETWORK 40
RollerDoor_1.TR_80_Deg := Trunnion_1.TR_80_Deg;

// NETWORK 41
RollerDoor_1.TT_0_Deg := TurnTable_1.TT_0_Deg;

// NETWORK 42
RollerDoor_1.TT_180_Deg := TurnTable_1.TT_180_Deg;

// NETWORK 43
RollerDoor_1(
    Roller_Up := RollerDoor_1.Roller_Up,
    Roller_Down := RollerDoor_1.Roller_Down,
    Part_Load_Comp := RollerDoor_1.Part_Load_Comp,
    Part_Unload_Comp := RollerDoor_1.Part_Unload_Comp,
    Weld_Comp := RollerDoor_1.Weld_Comp,
    TR_0_Deg := RollerDoor_1.TR_0_Deg,
    TR_50_Deg := RollerDoor_1.TR_50_Deg,
    TR_80_Deg := RollerDoor_1.TR_80_Deg,
    TT_0_Deg := RollerDoor_1.TT_0_Deg,
    TT_180_Deg := RollerDoor_1.TT_180_Deg); // RollerDoor

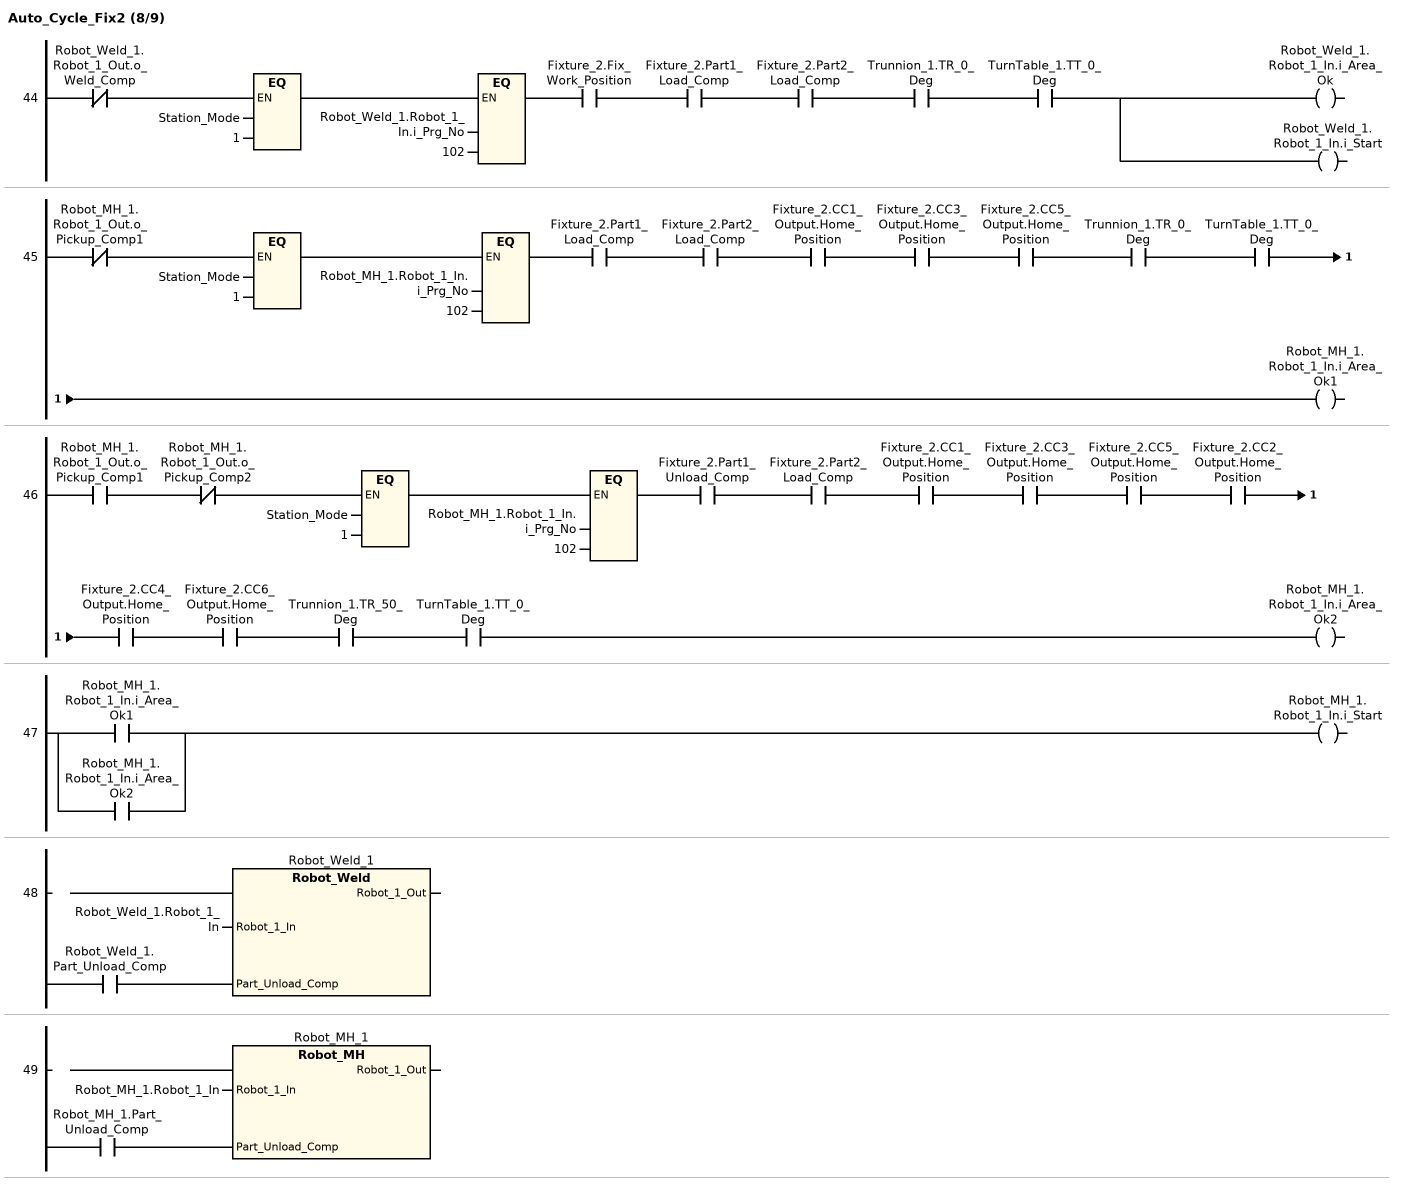
// NETWORK 44
_w1 := (NOT Robot_Weld_1.Robot_1_Out.o_Weld_Comp AND Station_Mode = 1 AND Robot_Weld_1.Robot_1_In.i_Prg_No = 102) AND Fixture_2.Fix_Work_Position AND Fixture_2.Part1_Load_Comp AND Fixture_2.Part2_Load_Comp AND Trunnion_1.TR_0_Deg AND TurnTable_1.TT_0_Deg;
Robot_Weld_1.Robot_1_In.i_Area_Ok := _w1;
Robot_Weld_1.Robot_1_In.i_Start := _w1;

// NETWORK 45
Robot_MH_1.Robot_1_In.i_Area_Ok1 := (NOT Robot_MH_1.Robot_1_Out.o_Pickup_Comp1 AND Station_Mode = 1 AND Robot_MH_1.Robot_1_In.i_Prg_No = 102) AND Fixture_2.Part1_Load_Comp AND Fixture_2.Part2_Load_Comp AND Fixture_2.CC1_Output.Home_Position AND Fixture_2.CC3_Output.Home_Position AND Fixture_2.CC5_Output.Home_Position AND Trunnion_1.TR_0_Deg AND TurnTable_1.TT_0_Deg;

// NETWORK 46
Robot_MH_1.Robot_1_In.i_Area_Ok2 := (Robot_MH_1.Robot_1_Out.o_Pickup_Comp1 AND NOT Robot_MH_1.Robot_1_Out.o_Pickup_Comp2 AND Station_Mode = 1 AND Robot_MH_1.Robot_1_In.i_Prg_No = 102) AND Fixture_2.Part1_Unload_Comp AND Fixture_2.Part2_Load_Comp AND Fixture_2.CC1_Output.Home_Position AND Fixture_2.CC3_Output.Home_Position AND Fixture_2.CC5_Output.Home_Position AND Fixture_2.CC2_Output.Home_Position AND Fixture_2.CC4_Output.Home_Position AND Fixture_2.CC6_Output.Home_Position AND Trunnion_1.TR_50_Deg AND TurnTable_1.TT_0_Deg;

// NETWORK 47
Robot_MH_1.Robot_1_In.i_Start := Robot_MH_1.Robot_1_In.i_Area_Ok1 OR Robot_MH_1.Robot_1_In.i_Area_Ok2;

// NETWORK 48
Robot_Weld_1(Robot_1_In := Robot_Weld_1.Robot_1_In, Part_Unload_Comp := Robot_Weld_1.Part_Unload_Comp); // Robot_Weld

// NETWORK 49
Robot_MH_1(Robot_1_In := Robot_MH_1.Robot_1_In, Part_Unload_Comp := Robot_MH_1.Part_Unload_Comp); // Robot_MH

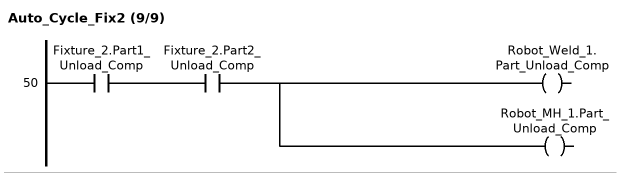
// NETWORK 50
_w2 := Fixture_2.Part1_Unload_Comp AND Fixture_2.Part2_Unload_Comp;
Robot_Weld_1.Part_Unload_Comp := _w2;
Robot_MH_1.Part_Unload_Comp := _w2;

END_PROGRAM

// ---- POUs/Fix2_FB.TcPOU
FUNCTION_BLOCK Fix2_FB
VAR_INPUT
CC1_Input 			: Fixture;					//Clamping Circuit-1
CC2_Input 			: Fixture;					//Clamping Circuit-2
CC3_Input 			: Fixture;					//Clamping Circuit-3
CC4_Input 			: Fixture;					//Clamping Circuit-4
CC5_Input 			: Fixture;					//Clamping Circuit-5
CC6_Input 			: Fixture;					//Clamping Circuit-6

Unit_Adv_Pb 		: BOOL;						//Fixture Cylinder Clamp Pb
Unit_Ret_Pb 		: BOOL;						//Fixture Cylinder Declamp Pb

Part1_Load_Comp 	: BOOL;						//OP710 Part-1 Load Complete
Part1_Unload_Comp 	: BOOL;						//OP710 Part-1 Unload Complete
Part2_Load_Comp 	: BOOL;						//OP710 Part-2 Load Complete
Part2_Unload_Comp 	: BOOL;						//OP710 Part-2 Unload Complete

Robot_Weld_Comp 	: BOOL;						//Robot Weld Complete
TR_0_Deg  			: BOOL;						//Trunnion at 0 degree
TR_20_Deg 			: BOOL;						//Trunnion at -20 degree
TR_50_Deg 			: BOOL;						//Trunnion at 50 degree

TT_180_Deg 			: BOOL;						//TurnTable at 180 degree
TT_0_Deg 			: BOOL;						//TurnTable at 0 degree
Roller_Down 		: BOOL;						//Roller Door Down position
Roller_Up 			: BOOL;						//Roller Door Up position
END_VAR

VAR_OUTPUT
CC1_Output 			: Fixture;							//Clamping Circuit-1
CC2_Output 			: Fixture;							//Clamping Circuit-2
CC3_Output 			: Fixture;							//Clamping Circuit-3
CC4_Output 			: Fixture;							//Clamping Circuit-4
CC5_Output 			: Fixture;							//Clamping Circuit-5
CC6_Output 			: Fixture;							//Clamping Circuit-6
Fix_Home_Position 	: BOOL;
Fix_Work_Position 	: BOOL;

END_VAR

VAR
Cyl_Delay 			: ARRAY [0..30] OF TON;
END_VAR

Fix_Home_Position := CC1_Output.Home_Position AND CC2_Output.Home_Position AND CC3_Output.Home_Position AND CC4_Output.Home_Position AND CC5_Output.Home_Position AND CC6_Output.Home_Position;
Fix_Work_Position := CC1_Output.Work_Position AND CC2_Output.Work_Position AND CC3_Output.Work_Position AND CC4_Output.Work_Position AND CC5_Output.Work_Position AND CC6_Output.Work_Position;

CASE Station_Mode OF
	
	0: 
	
	IF (CC5_Input.Manual_Sel AND Unit_Adv_Pb AND (NOT Unit_Ret_Pb) AND CC6_Output.Home_Position) THEN
		CC5_Output.o_Clamp_WP := TRUE;
		Cyl_Delay[0](IN:= CC5_Output.o_Clamp_WP, PT:= T#1S, Q=> , ET=> );
		IF Cyl_Delay[0].Q THEN
		CC5_Input.i_Clamp1_Fbk := CC5_Input.i_Clamp2_Fbk := CC5_Input.i_Clamp3_Fbk := CC5_Output.Work_Position := TRUE;
		CC5_Input.i_Declamp1_Fbk := CC5_Input.i_Declamp2_Fbk := CC5_Input.i_Declamp3_Fbk := CC5_Output.Home_Position := FALSE;
		CC5_Output.o_Clamp_WP := FALSE;
		END_IF
	ELSIF (CC5_Input.Manual_Sel AND Unit_Ret_Pb AND (NOT Unit_Adv_Pb) AND CC6_Output.Home_Position) THEN
		CC5_Output.o_Clamp_HP := TRUE;
		Cyl_Delay[1](IN:= CC5_Output.o_Clamp_HP, PT:= T#1S, Q=> , ET=> );
		IF Cyl_Delay[1].Q THEN
		CC5_Input.i_Declamp1_Fbk := CC5_Input.i_Declamp2_Fbk := CC5_Input.i_Declamp3_Fbk := CC5_Output.Home_Position := TRUE;
		CC5_Input.i_Clamp1_Fbk := CC5_Input.i_Clamp2_Fbk := CC5_Input.i_Clamp3_Fbk := CC5_Output.Work_Position := FALSE;
		CC5_Output.o_Clamp_HP := FALSE;
		END_IF
	END_IF
	
	IF (CC6_Input.Manual_Sel AND Unit_Adv_Pb AND (NOT Unit_Ret_Pb) AND CC5_Output.Work_Position) THEN
		CC6_Output.o_Clamp_WP := TRUE;
		Cyl_Delay[2](IN:= CC6_Output.o_Clamp_WP, PT:= T#1S, Q=> , ET=> );
		IF Cyl_Delay[2].Q THEN
		CC6_Input.i_Clamp1_Fbk := CC6_Input.i_Clamp2_Fbk := CC6_Input.i_Clamp3_Fbk := CC6_Output.Work_Position := TRUE;
		CC6_Input.i_Declamp1_Fbk := CC6_Input.i_Declamp2_Fbk := CC6_Input.i_Declamp3_Fbk := CC6_Output.Home_Position := FALSE;
		CC6_Output.o_Clamp_WP := FALSE;
		END_IF
	ELSIF (CC6_Input.Manual_Sel AND Unit_Ret_Pb AND (NOT Unit_Adv_Pb) AND CC5_Output.Work_Position) THEN
		CC6_Output.o_Clamp_HP := TRUE;
		Cyl_Delay[3](IN:= CC6_Output.o_Clamp_HP, PT:= T#1S, Q=> , ET=> );
		IF Cyl_Delay[3].Q THEN
		CC6_Input.i_Declamp1_Fbk := CC6_Input.i_Declamp2_Fbk := CC6_Input.i_Declamp3_Fbk := CC6_Output.Home_Position := TRUE;
		CC6_Input.i_Clamp1_Fbk := CC6_Input.i_Clamp2_Fbk := CC6_Input.i_Clamp3_Fbk := CC6_Output.Work_Position := FALSE;
		CC6_Output.o_Clamp_HP := FALSE;
		END_IF
	END_IF
	
	IF (CC1_Input.Manual_Sel AND Unit_Adv_Pb AND (NOT Unit_Ret_Pb) AND CC6_Output.Work_Position) THEN
		CC1_Output.o_Clamp_WP := TRUE;
		Cyl_Delay[4](IN:= CC1_Output.o_Clamp_WP, PT:= T#1S, Q=> , ET=> );
		IF Cyl_Delay[4].Q THEN
		CC1_Input.i_Clamp1_Fbk := CC1_Input.i_Clamp2_Fbk := CC1_Input.i_Clamp3_Fbk := CC1_Output.Work_Position := TRUE;
		CC1_Input.i_Declamp1_Fbk := CC1_Input.i_Declamp2_Fbk := CC1_Input.i_Declamp3_Fbk := CC1_Output.Home_Position := FALSE;
		CC1_Output.o_Clamp_WP := FALSE;
		END_IF
	ELSIF (CC1_Input.Manual_Sel AND Unit_Ret_Pb AND (NOT Unit_Adv_Pb) AND CC6_Output.Work_Position) THEN
		CC1_Output.o_Clamp_HP := TRUE;
		Cyl_Delay[5](IN:= CC1_Output.o_Clamp_HP, PT:= T#1S, Q=> , ET=> );
		IF Cyl_Delay[5].Q THEN
		CC1_Input.i_Declamp1_Fbk := CC1_Input.i_Declamp2_Fbk := CC1_Input.i_Declamp3_Fbk := CC1_Output.Home_Position := TRUE;
		CC1_Input.i_Clamp1_Fbk := CC1_Input.i_Clamp2_Fbk := CC1_Input.i_Clamp3_Fbk := CC1_Output.Work_Position := FALSE;
		CC1_Output.o_Clamp_HP := FALSE;
		END_IF
	END_IF
	
	IF (CC3_Input.Manual_Sel AND Unit_Adv_Pb AND (NOT Unit_Ret_Pb) AND CC1_Output.Work_Position) THEN
		CC3_Output.o_Clamp_WP := TRUE;
		Cyl_Delay[6](IN:= CC2_Output.o_Clamp_WP, PT:= T#1S, Q=> , ET=> );
		IF Cyl_Delay[6].Q THEN
		CC3_Input.i_Clamp1_Fbk := CC3_Input.i_Clamp2_Fbk := CC3_Input.i_Clamp3_Fbk := CC3_Output.Work_Position := TRUE;
		CC3_Input.i_Declamp1_Fbk := CC3_Input.i_Declamp2_Fbk := CC3_Input.i_Declamp3_Fbk := CC3_Output.Home_Position := FALSE;
		CC3_Output.o_Clamp_WP := FALSE;
		END_IF
	ELSIF (CC3_Input.Manual_Sel AND Unit_Ret_Pb AND (NOT Unit_Adv_Pb) AND CC1_Output.Work_Position) THEN
		CC3_Output.o_Clamp_HP := TRUE;
		Cyl_Delay[7](IN:= CC3_Output.o_Clamp_HP, PT:= T#1S, Q=> , ET=> );
		IF Cyl_Delay[7].Q THEN
		CC3_Input.i_Declamp1_Fbk := CC3_Input.i_Declamp2_Fbk := CC3_Input.i_Declamp3_Fbk := CC3_Output.Home_Position := TRUE;
		CC3_Input.i_Clamp1_Fbk := CC3_Input.i_Clamp2_Fbk := CC3_Input.i_Clamp3_Fbk := CC3_Output.Work_Position := FALSE;
		CC3_Output.o_Clamp_HP := FALSE;
		END_IF
	END_IF
	
	IF (CC2_Input.Manual_Sel AND Unit_Adv_Pb AND (NOT Unit_Ret_Pb) AND CC3_Output.Work_Position) THEN
		CC2_Output.o_Clamp_WP := TRUE;
		Cyl_Delay[8](IN:= CC2_Output.o_Clamp_WP, PT:= T#1S, Q=> , ET=> );
		IF Cyl_Delay[8].Q THEN
		CC2_Input.i_Clamp1_Fbk := CC2_Input.i_Clamp2_Fbk := CC2_Input.i_Clamp3_Fbk := CC2_Output.Work_Position := TRUE;
		CC2_Input.i_Declamp1_Fbk := CC2_Input.i_Declamp2_Fbk := CC2_Input.i_Declamp3_Fbk := CC2_Output.Home_Position := FALSE;
		CC2_Output.o_Clamp_WP := FALSE;
		END_IF
	ELSIF (CC2_Input.Manual_Sel AND Unit_Ret_Pb AND (NOT Unit_Adv_Pb) AND CC3_Output.Work_Position) THEN
		CC2_Output.o_Clamp_HP := TRUE;
		Cyl_Delay[9](IN:= CC2_Output.o_Clamp_HP, PT:= T#1S, Q=> , ET=> );
		IF Cyl_Delay[9].Q THEN
		CC2_Input.i_Declamp1_Fbk := CC2_Input.i_Declamp2_Fbk := CC2_Input.i_Declamp3_Fbk := CC2_Output.Home_Position := TRUE;
		CC2_Input.i_Clamp1_Fbk := CC2_Input.i_Clamp2_Fbk := CC2_Input.i_Clamp3_Fbk := CC2_Output.Work_Position := FALSE;
		CC2_Output.o_Clamp_HP := FALSE;
		END_IF
	END_IF
	
	IF (CC4_Input.Manual_Sel AND Unit_Adv_Pb AND (NOT Unit_Ret_Pb) AND CC2_Output.Work_Position) THEN
		CC4_Output.o_Clamp_WP := TRUE;
		Cyl_Delay[10](IN:= CC4_Output.o_Clamp_WP, PT:= T#1S, Q=> , ET=> );
		IF Cyl_Delay[10].Q THEN
		CC4_Input.i_Clamp1_Fbk := CC4_Input.i_Clamp2_Fbk := CC4_Input.i_Clamp3_Fbk := CC4_Output.Work_Position := TRUE;
		CC4_Input.i_Declamp1_Fbk := CC4_Input.i_Declamp2_Fbk := CC4_Input.i_Declamp3_Fbk := CC4_Output.Home_Position := FALSE;
		CC4_Output.o_Clamp_WP := FALSE;
		END_IF
	ELSIF (CC4_Input.Manual_Sel AND Unit_Ret_Pb AND (NOT Unit_Adv_Pb) AND CC2_Output.Work_Position) THEN
		CC4_Output.o_Clamp_HP := TRUE;
		Cyl_Delay[11](IN:= CC4_Output.o_Clamp_HP, PT:= T#1S, Q=> , ET=> );
		IF Cyl_Delay[11].Q THEN
		CC4_Input.i_Declamp1_Fbk := CC4_Input.i_Declamp2_Fbk := CC4_Input.i_Declamp3_Fbk := CC4_Output.Home_Position := TRUE;
		CC4_Input.i_Clamp1_Fbk := CC4_Input.i_Clamp2_Fbk := CC4_Input.i_Clamp3_Fbk := CC4_Output.Work_Position := FALSE;
		CC4_Output.o_Clamp_HP := FALSE;
		END_IF
	END_IF

	
	1:

	IF (Start_Pb AND CC5_Input.Auto_Sel AND TR_20_Deg AND Part1_Load_Comp AND CC6_Output.Home_Position) THEN
		CC5_Output.o_Clamp_WP := TRUE;
		Cyl_Delay[12](IN:= (CC5_Output.o_Clamp_WP), PT:= T#1S, Q=> , ET=> );
		IF Cyl_Delay[12].Q THEN
		CC5_Input.i_Declamp1_Fbk := CC5_Input.i_Declamp2_Fbk := CC5_Input.i_Declamp3_Fbk := CC5_Output.Home_Position := FALSE;
		CC5_Input.i_Clamp1_Fbk := CC5_Input.i_Clamp2_Fbk := CC5_Input.i_Clamp3_Fbk := CC5_Output.Work_Position := TRUE;
		CC5_Output.o_Clamp_WP := FALSE;
		END_IF
	END_IF
	IF (Start_Pb AND CC6_Input.Auto_Sel AND TR_20_Deg AND CC5_Output.Work_Position) THEN
		CC6_Output.o_Clamp_WP := TRUE;
		Cyl_Delay[13](IN:= CC6_Output.o_Clamp_WP, PT:= T#1S, Q=> , ET=> );
		IF Cyl_Delay[13].Q THEN
		CC6_Input.i_Declamp1_Fbk := CC6_Input.i_Declamp2_Fbk := CC6_Input.i_Declamp3_Fbk := CC6_Output.Home_Position := FALSE;
		CC6_Input.i_Clamp1_Fbk := CC6_Input.i_Clamp2_Fbk := CC6_Input.i_Clamp3_Fbk := CC6_Output.Work_Position := TRUE;
		CC6_Output.o_Clamp_WP := FALSE;
		END_IF
	END_IF
	IF (Start_Pb AND CC1_Input.Auto_Sel AND TR_20_Deg AND CC6_Output.Work_Position) THEN
		CC1_Output.o_Clamp_WP := TRUE;
		Cyl_Delay[14](IN:= CC1_Output.o_Clamp_WP, PT:= T#1S, Q=> , ET=> );
		IF Cyl_Delay[14].Q THEN
		CC1_Input.i_Declamp1_Fbk := CC1_Input.i_Declamp2_Fbk := CC1_Input.i_Declamp3_Fbk := CC1_Output.Home_Position := FALSE;
		CC1_Input.i_Clamp1_Fbk := CC1_Input.i_Clamp2_Fbk := CC1_Input.i_Clamp3_Fbk := CC1_Output.Work_Position := TRUE;
		CC1_Output.o_Clamp_WP := FALSE;
		END_IF
	END_IF
	IF (Start_Pb AND CC3_Input.Auto_Sel AND TR_20_Deg AND CC1_Output.Work_Position) THEN
		CC3_Output.o_Clamp_WP := TRUE;
		Cyl_Delay[14](IN:= CC3_Output.o_Clamp_WP, PT:= T#1S, Q=> , ET=> );
		IF Cyl_Delay[14].Q THEN
		CC3_Input.i_Declamp1_Fbk := CC3_Input.i_Declamp2_Fbk := CC3_Input.i_Declamp3_Fbk := CC3_Output.Home_Position := FALSE;
		CC3_Input.i_Clamp1_Fbk := CC3_Input.i_Clamp2_Fbk := CC3_Input.i_Clamp3_Fbk := CC3_Output.Work_Position := TRUE;
		CC3_Output.o_Clamp_WP := FALSE;
		END_IF
	END_IF
	IF (Start_Pb AND CC2_Input.Auto_Sel AND TR_50_Deg AND Part2_Load_Comp AND Roller_Down AND CC3_Output.Work_Position) THEN
		CC2_Output.o_Clamp_WP := TRUE;
		Cyl_Delay[15](IN:= CC2_Output.o_Clamp_WP, PT:= T#1S, Q=> , ET=> );
		IF Cyl_Delay[15].Q THEN
		CC2_Input.i_Declamp1_Fbk := CC2_Input.i_Declamp2_Fbk := CC2_Input.i_Declamp3_Fbk := CC2_Output.Home_Position := FALSE;
		CC2_Input.i_Clamp1_Fbk := CC2_Input.i_Clamp2_Fbk := CC2_Input.i_Clamp3_Fbk := CC2_Output.Work_Position := TRUE;
		CC2_Output.o_Clamp_WP := FALSE;
		END_IF
	END_IF
	IF (Start_Pb AND CC4_Input.Auto_Sel AND TR_50_Deg AND Roller_Down AND CC2_Output.Work_Position) THEN
		CC4_Output.o_Clamp_WP := TRUE;
		Cyl_Delay[16](IN:= CC4_Output.o_Clamp_WP, PT:= T#1S, Q=> , ET=> );
		IF Cyl_Delay[16].Q THEN
		CC4_Input.i_Declamp1_Fbk := CC4_Input.i_Declamp2_Fbk := CC4_Input.i_Declamp3_Fbk := CC4_Output.Home_Position := FALSE;
		CC4_Input.i_Clamp1_Fbk := CC4_Input.i_Clamp2_Fbk := CC4_Input.i_Clamp3_Fbk := CC4_Output.Work_Position := TRUE;
		CC4_Output.o_Clamp_WP := FALSE;
		END_IF
	END_IF
	
	IF (CC5_Input.Auto_Sel AND TT_0_Deg AND TR_0_Deg AND Robot_Weld_Comp) THEN
		CC5_Output.o_Clamp_HP := TRUE;
		Cyl_Delay[18](IN:= CC5_Output.o_Clamp_HP, PT:= T#1S, Q=> , ET=> );
		IF Cyl_Delay[18].Q THEN
		CC5_Input.i_Clamp1_Fbk := CC5_Input.i_Clamp2_Fbk := CC5_Input.i_Clamp3_Fbk := CC5_Output.Work_Position := FALSE;
		CC5_Input.i_Declamp1_Fbk := CC5_Input.i_Declamp2_Fbk := CC5_Input.i_Declamp3_Fbk := CC5_Output.Home_Position := TRUE;
		CC5_Output.o_clamp_HP := FALSE;
		END_IF
	END_IF
	IF (CC3_Input.Auto_Sel AND TT_0_Deg AND TR_0_Deg AND Robot_Weld_Comp) THEN
		CC3_Output.o_Clamp_HP := TRUE;
		Cyl_Delay[19](IN:= CC3_Output.o_Clamp_HP, PT:= T#1S, Q=> , ET=> );
		IF Cyl_Delay[19].Q THEN
		CC3_Input.i_Clamp1_Fbk := CC3_Input.i_Clamp2_Fbk := CC3_Input.i_Clamp3_Fbk := CC3_Output.Work_Position := FALSE;
		CC3_Input.i_Declamp1_Fbk := CC3_Input.i_Declamp2_Fbk := CC3_Input.i_Declamp3_Fbk := CC3_Output.Home_Position := TRUE;
		CC3_Output.o_clamp_HP := FALSE;
		END_IF
	END_IF
	IF (CC1_Input.Auto_Sel AND TT_0_Deg AND TR_0_Deg AND Robot_Weld_Comp) THEN
		CC1_Output.o_Clamp_HP := TRUE;
		Cyl_Delay[20](IN:= CC1_Output.o_Clamp_HP, PT:= T#1S, Q=> , ET=> );
		IF Cyl_Delay[20].Q THEN
		CC1_Input.i_Clamp1_Fbk := CC1_Input.i_Clamp2_Fbk := CC1_Input.i_Clamp3_Fbk := CC1_Output.Work_Position := FALSE;
		CC1_Input.i_Declamp1_Fbk := CC1_Input.i_Declamp2_Fbk := CC1_Input.i_Declamp3_Fbk := CC1_Output.Home_Position := TRUE;
		CC1_Output.o_clamp_HP := FALSE;
		END_IF
	END_IF
	IF (CC1_Output.Home_Position AND CC3_Output.Home_Position AND CC5_Output.Home_Position AND Roller_Up AND Part1_Unload_Comp AND TT_0_Deg AND TR_50_Deg AND Robot_Weld_Comp) THEN
		CC6_Output.o_Clamp_HP := TRUE;
		Cyl_Delay[21](IN:= CC6_Output.o_Clamp_HP, PT:= T#1S, Q=> , ET=> );
		IF Cyl_Delay[21].Q THEN
		CC6_Input.i_Clamp1_Fbk := CC6_Input.i_Clamp2_Fbk := CC6_Input.i_Clamp3_Fbk := CC6_Output.Work_Position := FALSE;
		CC6_Input.i_Declamp1_Fbk := CC6_Input.i_Declamp2_Fbk := CC6_Input.i_Declamp3_Fbk := CC6_Output.Home_Position := TRUE;
		CC6_Output.o_clamp_HP := FALSE;
		END_IF
	END_IF
	IF (CC6_Output.Home_Position AND Roller_Up AND Part1_Unload_Comp AND TT_0_Deg AND TR_50_Deg AND Robot_Weld_Comp) THEN
		CC4_Output.o_Clamp_HP := TRUE;
		Cyl_Delay[22](IN:= CC4_Output.o_Clamp_HP, PT:= T#1S, Q=> , ET=> );
		IF Cyl_Delay[22].Q THEN
		CC4_Input.i_Clamp1_Fbk := CC4_Input.i_Clamp2_Fbk := CC4_Input.i_Clamp3_Fbk := CC4_Output.Work_Position := FALSE;
		CC4_Input.i_Declamp1_Fbk := CC4_Input.i_Declamp2_Fbk := CC4_Input.i_Declamp3_Fbk := CC4_Output.Home_Position := TRUE;
		CC4_Output.o_clamp_HP := FALSE;
		END_IF
	END_IF
	IF (CC4_Output.Home_Position AND Roller_Up AND Part1_Unload_Comp AND TT_0_Deg AND TR_50_Deg AND Robot_Weld_Comp) THEN
		CC2_Output.o_Clamp_HP := TRUE;
		Cyl_Delay[23](IN:= CC2_Output.o_Clamp_HP, PT:= T#1S, Q=> , ET=> );
		IF Cyl_Delay[23].Q THEN
		CC2_Input.i_Clamp1_Fbk := CC2_Input.i_Clamp2_Fbk := CC2_Input.i_Clamp3_Fbk := CC2_Output.Work_Position := FALSE;
		CC2_Input.i_Declamp1_Fbk := CC2_Input.i_Declamp2_Fbk := CC2_Input.i_Declamp3_Fbk := CC2_Output.Home_Position := TRUE;
		CC2_Output.o_clamp_HP := FALSE;
		END_IF
	END_IF

END_CASE

END_FUNCTION_BLOCK

// ---- GlobalTextList.TcGTLO
TEXTLIST GlobalTextList
  593 = '%2f'
  846 = 'Auto'
  758 = 'Auto/Manual'
  319 = 'CC1'
  821 = 'CC2'
  275 = 'CC3'
  146 = 'CC4'
  865 = 'CC5'
  143 = 'CC6'
  155 = 'Clamp'
  609 = 'Declamp'
  765 = 'Estop OK'
  659 = 'Fault Reset'
  46 = 'Home Pos.'
  907 = 'Manual'
  47 = 'Master On'
  610 = 'MH Robot'
  256 = 'Part-1 Load'
  70 = 'Part-1 Load Comp'
  50 = 'Part-1 Unload Comp'
  790 = 'Part-2 Load'
  687 = 'Part-2 Load Comp'
  700 = 'Part-2 Unload Comp'
  753 = 'Pickup Area-1 OK'
  147 = 'Pickup Area-2 OK'
  480 = 'Pickup Comp.-1'
  835 = 'Pickup Comp.-2'
  464 = 'Roller Door Down'
  915 = 'Roller Door Up'
  399 = 'Safety OK'
  844 = 'Start'
  82 = 'Trunnion -20 Deg'
  384 = 'Trunnion 0 Deg'
  396 = 'Trunnion 45 Deg'
  760 = 'Trunnion 50 Deg'
  655 = 'Trunnion 80 Deg'
  518 = 'TurnTable 0 Deg'
  139 = 'TurnTable 180 Deg'
  253 = 'Weld Area OK'
  786 = 'Weld Comp.'
  966 = 'Weld Robot'
END_TEXTLIST

// ---- VISUs/Auto_Cycle_Fix1.TcVIS
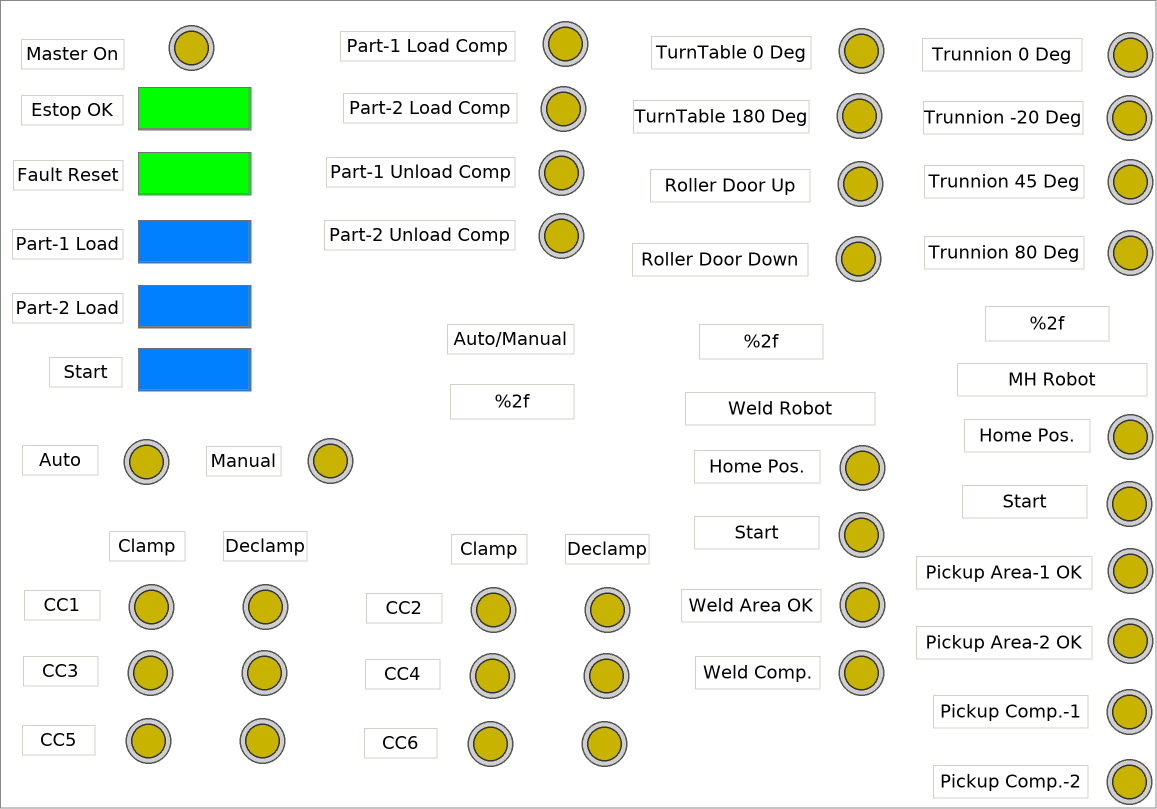
VISUALIZATION Auto_Cycle_Fix1  // 1157x809
    Lamp1 (539,17 53x54), variable: Auto_Cycle_Fix1.Fixture_1.Part1_Load_Comp, style: Lamp-Lamp1-Yellow
    Textfield (340,31 175x30), "Part-1 Load Comp"
    Textfield (343,93 174x30), "Part-2 Load Comp"
    Lamp1 (537,82 53x54), variable: Auto_Cycle_Fix1.Fixture_1.Part2_Load_Comp, style: Lamp-Lamp1-Yellow
    Textfield (651,36 160x33), "TurnTable 0 Deg"
    Lamp1 (835,24 53x54), variable: Auto_Cycle_Fix1.TurnTable_0.TT_0_Deg, style: Lamp-Lamp1-Yellow
    Textfield (633,100 176x33), "TurnTable 180 Deg"
    Lamp1 (833,89 53x54), variable: Auto_Cycle_Fix1.TurnTable_0.TT_180_Deg, style: Lamp-Lamp1-Yellow
    Textfield (922,38 160x33), "Trunnion 0 Deg"
    Lamp1 (1104,28 53x54), variable: Auto_Cycle_Fix1.Trunnion_0.TR_0_Deg, style: Lamp-Lamp1-Yellow
    Textfield (923,101 160x33), "Trunnion -20 Deg"
    Lamp1 (1103,91 53x54), variable: Auto_Cycle_Fix1.Trunnion_0.TR_20_Deg, style: Lamp-Lamp1-Yellow
    Lamp1 (1104,155 53x54), variable: Auto_Cycle_Fix1.Trunnion_0.TR_45_Deg, style: Lamp-Lamp1-Yellow
    Textfield (924,165 160x33), "Trunnion 45 Deg"
    Lamp1 (1104,226 53x54), variable: Auto_Cycle_Fix1.Trunnion_0.TR_80_Deg, style: Lamp-Lamp1-Yellow
    Textfield (924,236 160x33), "Trunnion 80 Deg"
    Textfield (24,590 76x30), "CC1"
    Textfield (23,656 75x30), "CC3"
    Textfield (22,725 73x30), "CC5"
    Lamp1 (125,580 53x54), variable: Auto_Cycle_Fix1.Fixture_1.CC1_Output.Work_Position, style: Lamp-Lamp1-Yellow
    Lamp1 (124,646 53x54), variable: Auto_Cycle_Fix1.Fixture_1.CC3_Output.Work_Position, style: Lamp-Lamp1-Yellow
    Lamp1 (122,714 53x54), variable: Auto_Cycle_Fix1.Fixture_1.CC5_Output.Work_Position, style: Lamp-Lamp1-Yellow
    Textfield (109,531 76x30), "Clamp"
    Lamp1 (239,580 53x54), variable: Auto_Cycle_Fix1.Fixture_1.CC1_Output.Home_Position, style: Lamp-Lamp1-Yellow
    Lamp1 (238,646 53x54), variable: Auto_Cycle_Fix1.Fixture_1.CC3_Output.Home_Position, style: Lamp-Lamp1-Yellow
    Lamp1 (236,714 53x54), variable: Auto_Cycle_Fix1.Fixture_1.CC5_Output.Home_Position, style: Lamp-Lamp1-Yellow
    Textfield (223,531 84x30), "Declamp"
    Textfield (366,593 76x30), "CC2"
    Textfield (365,659 75x30), "CC4"
    Textfield (364,728 73x30), "CC6"
    Lamp1 (467,583 53x54), variable: Auto_Cycle_Fix1.Fixture_1.CC2_Output.Work_Position, style: Lamp-Lamp1-Yellow
    Lamp1 (466,649 53x54), variable: Auto_Cycle_Fix1.Fixture_1.CC4_Output.Work_Position, style: Lamp-Lamp1-Yellow
    Lamp1 (464,717 53x54), variable: Auto_Cycle_Fix1.Fixture_1.CC6_Output.Work_Position, style: Lamp-Lamp1-Yellow
    Textfield (451,534 76x30), "Clamp"
    Lamp1 (581,583 53x54), variable: Auto_Cycle_Fix1.Fixture_1.CC2_Output.Home_Position, style: Lamp-Lamp1-Yellow
    Lamp1 (580,649 53x54), variable: Auto_Cycle_Fix1.Fixture_1.CC4_Output.Home_Position, style: Lamp-Lamp1-Yellow
    Lamp1 (578,717 53x54), variable: Auto_Cycle_Fix1.Fixture_1.CC6_Output.Home_Position, style: Lamp-Lamp1-Yellow
    Textfield (565,534 84x30), "Declamp"
    Textfield (22,445 76x30), "Auto"
    Textfield (206,446 75x30), "Manual"
    Lamp1 (304,434 53x54), variable: Manual_Mode, style: Lamp-Lamp1-Yellow
    Textfield (650,169 160x33), "Roller Door Up"
    Lamp1 (834,157 53x54), variable: Auto_Cycle_Fix1.RollerDoor_0.Roller_Up, style: Lamp-Lamp1-Yellow
    Textfield (632,243 176x33), "Roller Door Down"
    Lamp1 (832,232 53x54), variable: Auto_Cycle_Fix1.RollerDoor_0.Roller_Down, style: Lamp-Lamp1-Yellow
    Textfield (694,450 126x33), "Home Pos."
    Lamp1 (836,441 53x54), variable: Auto_Cycle_Fix1.Robot_Weld_0.Robot_1_In.i_Home, style: Lamp-Lamp1-Yellow
    Textfield (681,589 140x33), "Weld Area OK"
    Lamp1 (836,578 53x54), variable: Auto_Cycle_Fix1.Robot_Weld_0.Robot_1_In.i_Area_Ok, style: Lamp-Lamp1-Yellow
    Textfield (695,656 125x33), "Weld Comp."
    Lamp1 (835,646 53x54), variable: Auto_Cycle_Fix1.Robot_Weld_0.Robot_1_Out.o_Weld_Comp, style: Lamp-Lamp1-Yellow
    Textfield (685,392 190x33), "Weld Robot"
    Textfield (957,363 190x33), "MH Robot"
    Textfield (694,516 125x33), "Start"
    Lamp1 (835,508 53x54), variable: Auto_Cycle_Fix1.Robot_Weld_0.Robot_1_In.i_Start, style: Lamp-Lamp1-Yellow
    Textfield (964,419 126x33), "Home Pos."
    Lamp1 (1104,410 53x54), variable: Auto_Cycle_Fix1.Robot_MH_0.Robot_1_In.i_Home, style: Lamp-Lamp1-Yellow
    Textfield (916,556 176x33), "Pickup Area-1 OK"
    Lamp1 (1104,544 53x54), variable: Auto_Cycle_Fix1.Robot_MH_0.Robot_1_In.i_Area_Ok1, style: Lamp-Lamp1-Yellow
    Textfield (933,695 155x33), "Pickup Comp.-1"
    Lamp1 (1103,685 53x54), variable: Auto_Cycle_Fix1.Robot_MH_0.Robot_1_Out.o_Pickup_Comp1, style: Lamp-Lamp1-Yellow
    Textfield (962,485 125x33), "Start"
    Lamp1 (1103,477 53x54), variable: Auto_Cycle_Fix1.Robot_MH_0.Robot_1_In.i_Start, style: Lamp-Lamp1-Yellow
    Textfield (12,229 111x30), "Part-1 Load"
    Button (138,220 113x43)
        p573394764: Fix1_Part_1_Load
        toggle Fix1_Part_1_Load
    Textfield (447,324 127x30), "Auto/Manual"
    Textfield (326,157 189x30), "Part-1 Unload Comp"
    Lamp1 (535,146 53x54), variable: Auto_Cycle_Fix1.Fixture_1.Part1_Unload_Comp, style: Lamp-Lamp1-Yellow
    Textfield (324,220 191x30), "Part-2 Unload Comp"
    Lamp1 (535,209 53x54), variable: Auto_Cycle_Fix1.Fixture_1.Part2_Unload_Comp, style: Lamp-Lamp1-Yellow
    Textfield (450,384 124x35), "%2f", text variable: Station_Mode
        OnMouseDown: write Station_Mode via VisuDialogs.Numpad
    Textfield (916,626 176x33), "Pickup Area-2 OK"
    Lamp1 (1104,614 53x54), variable: Auto_Cycle_Fix1.Robot_MH_0.Robot_1_In.i_Area_Ok2, style: Lamp-Lamp1-Yellow
    Textfield (933,765 155x33), "Pickup Comp.-2"
    Lamp1 (1103,755 53x54), variable: Auto_Cycle_Fix1.Robot_MH_0.Robot_1_Out.o_Pickup_Comp2, style: Lamp-Lamp1-Yellow
    Lamp1 (120,435 53x54), variable: Auto_Mode, style: Lamp-Lamp1-Yellow
    Textfield (21,39 103x30), "Master On"
    Button (138,152 113x43)
        p573394764: Fault_Reset
        tap Fault_Reset
    Textfield (13,160 110x30), "Fault Reset"
    Textfield (12,293 111x30), "Part-2 Load"
    Button (138,285 113x43)
        p573394764: Fix1_Part_2_Load
        toggle Fix1_Part_2_Load
    Textfield (49,357 73x30), "Start"
    Button (138,348 113x43)
        p573394764: Start_Pb
        tap Start_Pb
    Textfield (699,324 124x35), "%2f", text variable: Auto_Cycle_Fix1.Robot_Weld_0.Robot_1_In.i_Prg_No
        OnMouseDown: write Auto_Cycle_Fix1.Robot_Weld_0.Robot_1_In.i_Prg_No via VisuDialogs.Numpad
    Textfield (985,306 124x35), "%2f", text variable: Auto_Cycle_Fix1.Robot_MH_0.Robot_1_In.i_Prg_No
        OnMouseDown: write Auto_Cycle_Fix1.Robot_MH_0.Robot_1_In.i_Prg_No via VisuDialogs.Numpad
    Lamp1 (165,21 53x54), variable: Master_On, style: Lamp-Lamp1-Yellow
    Button (138,87 113x43)
        p573394764: EStop
        toggle EStop
    Textfield (21,95 102x30), "Estop OK"
END_VISUALIZATION

// ---- VISUs/Auto_Cycle_Fix2.TcVIS
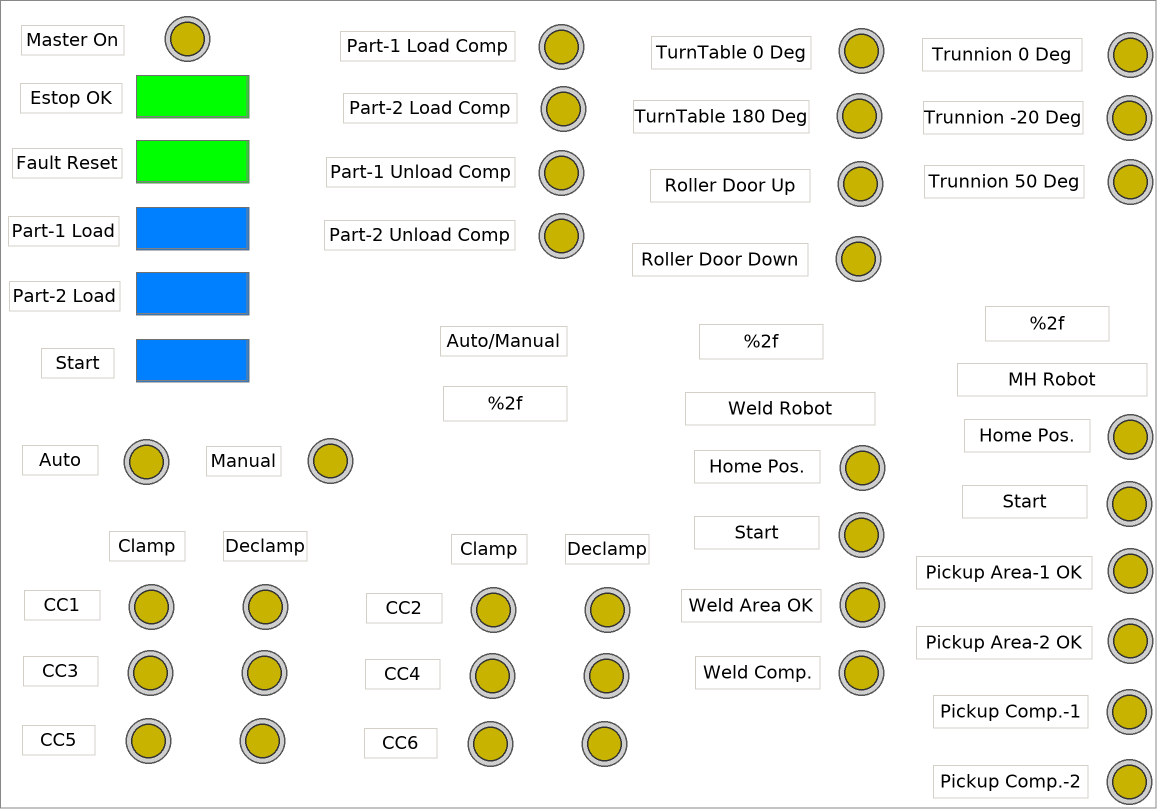
VISUALIZATION Auto_Cycle_Fix2  // 1157x809
    Textfield (340,31 175x30), "Part-1 Load Comp"
    Textfield (343,93 174x30), "Part-2 Load Comp"
    Lamp1 (537,82 53x54), variable: Auto_Cycle_Fix2.Fixture_2.Part2_Load_Comp, style: Lamp-Lamp1-Yellow
    Textfield (651,36 160x33), "TurnTable 0 Deg"
    Lamp1 (835,24 53x54), variable: Auto_Cycle_Fix2.TurnTable_1.TT_0_Deg, style: Lamp-Lamp1-Yellow
    Textfield (633,100 176x33), "TurnTable 180 Deg"
    Lamp1 (833,89 53x54), variable: Auto_Cycle_Fix2.TurnTable_1.TT_180_Deg, style: Lamp-Lamp1-Yellow
    Textfield (922,38 160x33), "Trunnion 0 Deg"
    Lamp1 (1104,28 53x54), variable: Auto_Cycle_Fix2.Trunnion_1.TR_0_Deg, style: Lamp-Lamp1-Yellow
    Textfield (923,101 160x33), "Trunnion -20 Deg"
    Lamp1 (1103,91 53x54), variable: Auto_Cycle_Fix2.Trunnion_1.TR_20_Deg, style: Lamp-Lamp1-Yellow
    Lamp1 (1104,155 53x54), variable: Auto_Cycle_Fix2.Trunnion_1.TR_50_Deg, style: Lamp-Lamp1-Yellow
    Textfield (924,165 160x33), "Trunnion 50 Deg"
    Textfield (24,590 76x30), "CC1"
    Textfield (23,656 75x30), "CC3"
    Textfield (22,725 73x30), "CC5"
    Lamp1 (125,580 53x54), variable: Auto_Cycle_Fix2.Fixture_2.CC1_Output.Work_Position, style: Lamp-Lamp1-Yellow
    Lamp1 (124,646 53x54), variable: Auto_Cycle_Fix2.Fixture_2.CC3_Output.Work_Position, style: Lamp-Lamp1-Yellow
    Lamp1 (122,714 53x54), variable: Auto_Cycle_Fix2.Fixture_2.CC5_Output.Work_Position, style: Lamp-Lamp1-Yellow
    Textfield (109,531 76x30), "Clamp"
    Lamp1 (239,580 53x54), variable: Auto_Cycle_Fix2.Fixture_2.CC1_Output.Home_Position, style: Lamp-Lamp1-Yellow
    Lamp1 (238,646 53x54), variable: Auto_Cycle_Fix2.Fixture_2.CC3_Output.Home_Position, style: Lamp-Lamp1-Yellow
    Lamp1 (236,714 53x54), variable: Auto_Cycle_Fix2.Fixture_2.CC5_Output.Home_Position, style: Lamp-Lamp1-Yellow
    Textfield (223,531 84x30), "Declamp"
    Textfield (366,593 76x30), "CC2"
    Textfield (365,659 75x30), "CC4"
    Textfield (364,728 73x30), "CC6"
    Lamp1 (467,583 53x54), variable: Auto_Cycle_Fix2.Fixture_2.CC2_Output.Work_Position, style: Lamp-Lamp1-Yellow
    Lamp1 (466,649 53x54), variable: Auto_Cycle_Fix2.Fixture_2.CC4_Output.Work_Position, style: Lamp-Lamp1-Yellow
    Lamp1 (464,717 53x54), variable: Auto_Cycle_Fix2.Fixture_2.CC6_Output.Work_Position, style: Lamp-Lamp1-Yellow
    Textfield (451,534 76x30), "Clamp"
    Lamp1 (581,583 53x54), variable: Auto_Cycle_Fix2.Fixture_2.CC2_Output.Home_Position, style: Lamp-Lamp1-Yellow
    Lamp1 (580,649 53x54), variable: Auto_Cycle_Fix2.Fixture_2.CC4_Output.Home_Position, style: Lamp-Lamp1-Yellow
    Lamp1 (578,717 53x54), variable: Auto_Cycle_Fix2.Fixture_2.CC6_Output.Home_Position, style: Lamp-Lamp1-Yellow
    Textfield (565,534 84x30), "Declamp"
    Textfield (22,445 76x30), "Auto"
    Textfield (206,446 75x30), "Manual"
    Lamp1 (304,434 53x54), variable: Manual_Mode, style: Lamp-Lamp1-Yellow
    Textfield (650,169 160x33), "Roller Door Up"
    Lamp1 (834,157 53x54), variable: Auto_Cycle_Fix2.RollerDoor_1.Roller_Up, style: Lamp-Lamp1-Yellow
    Textfield (632,243 176x33), "Roller Door Down"
    Lamp1 (832,232 53x54), variable: Auto_Cycle_Fix2.RollerDoor_1.Roller_Down, style: Lamp-Lamp1-Yellow
    Textfield (694,450 126x33), "Home Pos."
    Lamp1 (836,441 53x54), variable: Auto_Cycle_Fix2.Robot_Weld_1.Robot_1_In.i_Home, style: Lamp-Lamp1-Yellow
    Textfield (681,589 140x33), "Weld Area OK"
    Lamp1 (836,578 53x54), variable: Auto_Cycle_Fix2.Robot_Weld_1.Robot_1_In.i_Area_Ok, style: Lamp-Lamp1-Yellow
    Textfield (695,656 125x33), "Weld Comp."
    Lamp1 (835,646 53x54), variable: Auto_Cycle_Fix2.Robot_Weld_1.Robot_1_Out.o_Weld_Comp, style: Lamp-Lamp1-Yellow
    Textfield (685,392 190x33), "Weld Robot"
    Textfield (957,363 190x33), "MH Robot"
    Textfield (694,516 125x33), "Start"
    Lamp1 (835,508 53x54), variable: Auto_Cycle_Fix2.Robot_Weld_1.Robot_1_In.i_Start, style: Lamp-Lamp1-Yellow
    Textfield (964,419 126x33), "Home Pos."
    Lamp1 (1104,410 53x54), variable: Auto_Cycle_Fix2.Robot_MH_1.Robot_1_In.i_Home, style: Lamp-Lamp1-Yellow
    Textfield (916,556 176x33), "Pickup Area-1 OK"
    Lamp1 (1104,544 53x54), variable: Auto_Cycle_Fix2.Robot_MH_1.Robot_1_In.i_Area_Ok1, style: Lamp-Lamp1-Yellow
    Textfield (933,695 155x33), "Pickup Comp.-1"
    Lamp1 (1103,685 53x54), variable: Auto_Cycle_Fix2.Robot_MH_1.Robot_1_Out.o_Pickup_Comp1, style: Lamp-Lamp1-Yellow
    Textfield (962,485 125x33), "Start"
    Lamp1 (1103,477 53x54), variable: Auto_Cycle_Fix2.Robot_MH_1.Robot_1_In.i_Start, style: Lamp-Lamp1-Yellow
    Textfield (8,216 111x30), "Part-1 Load"
    Button (136,207 113x43)
        p573394764: Fix2_Part_1_Load
        toggle Fix2_Part_1_Load
    Textfield (440,326 127x30), "Auto/Manual"
    Textfield (326,157 189x30), "Part-1 Unload Comp"
    Lamp1 (535,146 53x54), variable: Auto_Cycle_Fix2.Fixture_2.Part1_Unload_Comp, style: Lamp-Lamp1-Yellow
    Textfield (324,220 191x30), "Part-2 Unload Comp"
    Lamp1 (535,209 53x54), variable: Auto_Cycle_Fix2.Fixture_2.Part2_Unload_Comp, style: Lamp-Lamp1-Yellow
    Textfield (443,386 124x35), "%2f", text variable: Station_Mode
        OnMouseDown: write Station_Mode via VisuDialogs.Numpad
    Textfield (916,626 176x33), "Pickup Area-2 OK"
    Lamp1 (1104,614 53x54), variable: Auto_Cycle_Fix2.Robot_MH_1.Robot_1_In.i_Area_Ok2, style: Lamp-Lamp1-Yellow
    Textfield (933,765 155x33), "Pickup Comp.-2"
    Lamp1 (1103,755 53x54), variable: Auto_Cycle_Fix2.Robot_MH_1.Robot_1_Out.o_Pickup_Comp2, style: Lamp-Lamp1-Yellow
    Lamp1 (120,435 53x54), variable: Auto_Mode, style: Lamp-Lamp1-Yellow
    Textfield (9,281 111x30), "Part-2 Load"
    Button (136,272 113x43)
        p573394764: Fix2_Part_2_Load
        toggle Fix2_Part_2_Load
    Textfield (41,348 73x30), "Start"
    Button (136,339 113x43)
        p573394764: Start_Pb
        tap Start_Pb
    Textfield (699,324 124x35), "%2f", text variable: Auto_Cycle_Fix2.Robot_Weld_1.Robot_1_In.i_Prg_No
        OnMouseDown: write Auto_Cycle_Fix2.Robot_Weld_1.Robot_1_In.i_Prg_No via VisuDialogs.Numpad
    Textfield (985,306 124x35), "%2f", text variable: Auto_Cycle_Fix2.Robot_MH_1.Robot_1_In.i_Prg_No
        OnMouseDown: write Auto_Cycle_Fix2.Robot_MH_1.Robot_1_In.i_Prg_No via VisuDialogs.Numpad
    Lamp1 (535,20 53x54), variable: Auto_Cycle_Fix2.Fixture_2.Part1_Load_Comp, style: Lamp-Lamp1-Yellow
    Textfield (21,25 103x30), "Master On"
    Button (136,140 113x43)
        p573394764: Fault_Reset
        tap Fault_Reset
    Textfield (12,148 110x30), "Fault Reset"
    Lamp1 (161,12 53x54), variable: Master_On, style: Lamp-Lamp1-Yellow
    Button (136,75 113x43)
        p573394764: EStop
        toggle EStop
    Textfield (20,83 102x30), "Estop OK"
END_VISUALIZATION

// ---- VISUs/Manual_Action_Fix1.TcVIS
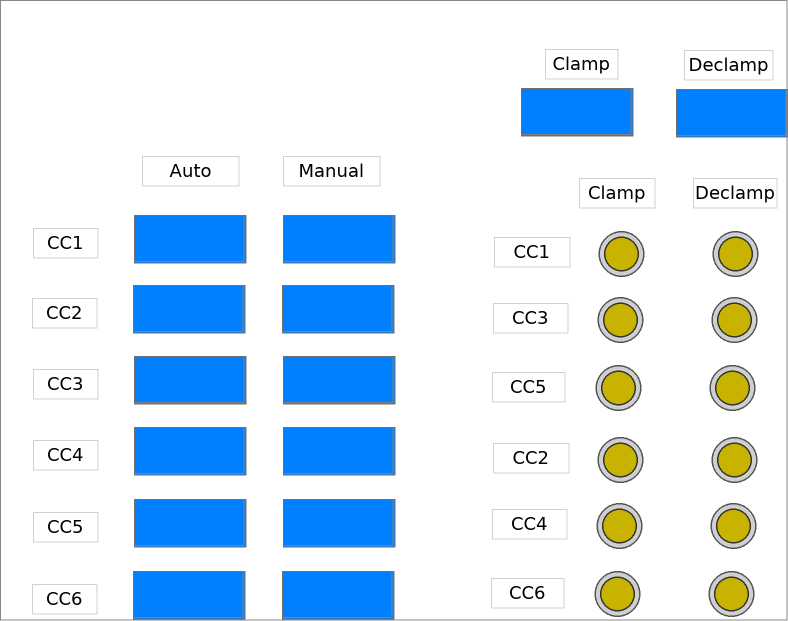
VISUALIZATION Manual_Action_Fix1  // 788x621
    Textfield (142,156 97x30), "Auto"
    Textfield (545,49 73x30), "Clamp"
    Button (521,88 112x48)
        p573394764: Auto_Cycle_Fix1.Fixture_1.Unit_Adv_Pb
        tap Auto_Cycle_Fix1.Fixture_1.Unit_Adv_Pb
    Textfield (684,50 89x30), "Declamp"
    Button (676,89 112x48)
        p573394764: Auto_Cycle_Fix1.Fixture_1.Unit_Ret_Pb
        tap Auto_Cycle_Fix1.Fixture_1.Unit_Ret_Pb
    Textfield (494,237 76x30), "CC1"
    Textfield (493,303 75x30), "CC3"
    Textfield (492,372 73x30), "CC5"
    Lamp1 (595,227 53x54), variable: Auto_Cycle_Fix1.Fixture_1.CC1_Output.Work_Position, style: Lamp-Lamp1-Yellow
    Lamp1 (594,293 53x54), variable: Auto_Cycle_Fix1.Fixture_1.CC3_Output.Work_Position, style: Lamp-Lamp1-Yellow
    Lamp1 (592,361 53x54), variable: Auto_Cycle_Fix1.Fixture_1.CC5_Output.Work_Position, style: Lamp-Lamp1-Yellow
    Textfield (579,178 76x30), "Clamp"
    Lamp1 (709,227 53x54), variable: Auto_Cycle_Fix1.Fixture_1.CC1_Output.Home_Position, style: Lamp-Lamp1-Yellow
    Lamp1 (708,293 53x54), variable: Auto_Cycle_Fix1.Fixture_1.CC3_Output.Home_Position, style: Lamp-Lamp1-Yellow
    Lamp1 (706,361 53x54), variable: Auto_Cycle_Fix1.Fixture_1.CC5_Output.Home_Position, style: Lamp-Lamp1-Yellow
    Textfield (693,178 84x30), "Declamp"
    Textfield (493,443 76x30), "CC2"
    Textfield (492,509 75x30), "CC4"
    Textfield (491,578 73x30), "CC6"
    Lamp1 (594,433 53x54), variable: Auto_Cycle_Fix1.Fixture_1.CC2_Output.Work_Position, style: Lamp-Lamp1-Yellow
    Lamp1 (593,499 53x54), variable: Auto_Cycle_Fix1.Fixture_1.CC4_Output.Work_Position, style: Lamp-Lamp1-Yellow
    Lamp1 (591,567 53x54), variable: Auto_Cycle_Fix1.Fixture_1.CC6_Output.Work_Position, style: Lamp-Lamp1-Yellow
    Lamp1 (708,433 53x54), variable: Auto_Cycle_Fix1.Fixture_1.CC2_Output.Home_Position, style: Lamp-Lamp1-Yellow
    Lamp1 (707,499 53x54), variable: Auto_Cycle_Fix1.Fixture_1.CC4_Output.Home_Position, style: Lamp-Lamp1-Yellow
    Lamp1 (705,567 53x54), variable: Auto_Cycle_Fix1.Fixture_1.CC6_Output.Home_Position, style: Lamp-Lamp1-Yellow
    Button (134,215 112x48)
        p573394764: Auto_Cycle_Fix1.Fixture_1.CC1_Input.Auto_Sel
        toggle Auto_Cycle_Fix1.Fixture_1.CC1_Input.Auto_Sel
    Textfield (33,228 65x30), "CC1"
    Button (133,285 112x48)
        p573394764: Auto_Cycle_Fix1.Fixture_1.CC2_Input.Auto_Sel
        toggle Auto_Cycle_Fix1.Fixture_1.CC2_Input.Auto_Sel
    Textfield (32,298 65x30), "CC2"
    Button (134,356 112x48)
        p573394764: Auto_Cycle_Fix1.Fixture_1.CC3_Input.Auto_Sel
        toggle Auto_Cycle_Fix1.Fixture_1.CC3_Input.Auto_Sel
    Textfield (33,369 65x30), "CC3"
    Button (134,427 112x48)
        p573394764: Auto_Cycle_Fix1.Fixture_1.CC4_Input.Auto_Sel
        toggle Auto_Cycle_Fix1.Fixture_1.CC4_Input.Auto_Sel
    Textfield (33,440 65x30), "CC4"
    Button (134,499 112x48)
        p573394764: Auto_Cycle_Fix1.Fixture_1.CC5_Input.Auto_Sel
        toggle Auto_Cycle_Fix1.Fixture_1.CC5_Input.Auto_Sel
    Textfield (33,512 65x30), "CC5"
    Button (133,571 112x48)
        p573394764: Auto_Cycle_Fix1.Fixture_1.CC6_Input.Auto_Sel
        toggle Auto_Cycle_Fix1.Fixture_1.CC6_Input.Auto_Sel
    Textfield (32,584 65x30), "CC6"
    Button (283,215 112x48)
        p573394764: Auto_Cycle_Fix1.Fixture_1.CC1_Input.Manual_Sel
        toggle Auto_Cycle_Fix1.Fixture_1.CC1_Input.Manual_Sel
    Button (282,285 112x48)
        p573394764: Auto_Cycle_Fix1.Fixture_1.CC2_Input.Manual_Sel
        toggle Auto_Cycle_Fix1.Fixture_1.CC2_Input.Manual_Sel
    Button (283,356 112x48)
        p573394764: Auto_Cycle_Fix1.Fixture_1.CC3_Input.Manual_Sel
        toggle Auto_Cycle_Fix1.Fixture_1.CC3_Input.Manual_Sel
    Button (283,427 112x48)
        p573394764: Auto_Cycle_Fix1.Fixture_1.CC4_Input.Manual_Sel
        toggle Auto_Cycle_Fix1.Fixture_1.CC4_Input.Manual_Sel
    Button (283,499 112x48)
        p573394764: Auto_Cycle_Fix1.Fixture_1.CC5_Input.Manual_Sel
        toggle Auto_Cycle_Fix1.Fixture_1.CC5_Input.Manual_Sel
    Button (282,571 112x48)
        p573394764: Auto_Cycle_Fix1.Fixture_1.CC6_Input.Manual_Sel
        toggle Auto_Cycle_Fix1.Fixture_1.CC6_Input.Manual_Sel
    Textfield (283,156 97x30), "Manual"
END_VISUALIZATION

// ---- VISUs/Manual_Action_Fix2.TcVIS
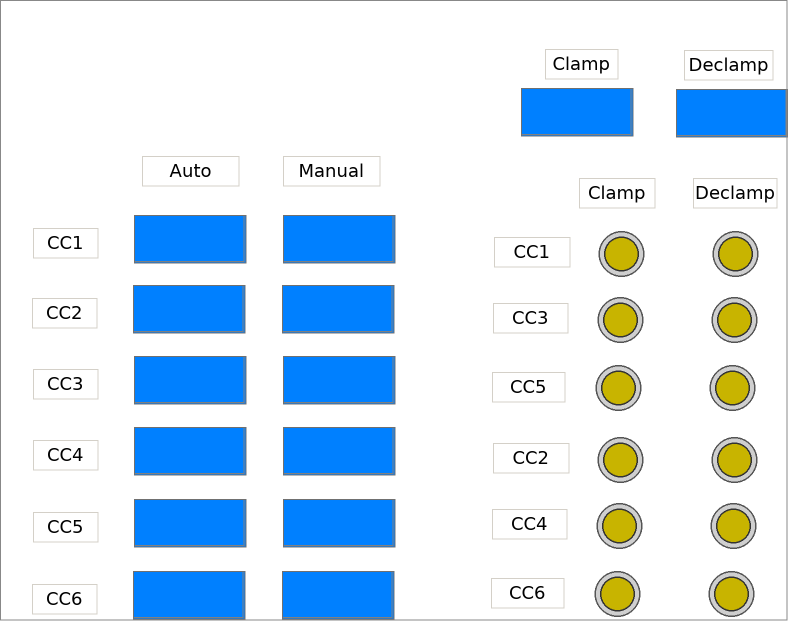
VISUALIZATION Manual_Action_Fix2  // 788x621
    Textfield (142,156 97x30), "Auto"
    Textfield (545,49 73x30), "Clamp"
    Button (521,88 112x48)
        p573394764: Auto_Cycle_Fix2.Fixture_2.Unit_Adv_Pb
        tap Auto_Cycle_Fix2.Fixture_2.Unit_Adv_Pb
    Textfield (684,50 89x30), "Declamp"
    Button (676,89 112x48)
        p573394764: Auto_Cycle_Fix2.Fixture_2.Unit_Ret_Pb
        tap Auto_Cycle_Fix2.Fixture_2.Unit_Ret_Pb
    Textfield (494,237 76x30), "CC1"
    Textfield (493,303 75x30), "CC3"
    Textfield (492,372 73x30), "CC5"
    Lamp1 (595,227 53x54), variable: Auto_Cycle_Fix2.Fixture_2.CC1_Output.Work_Position, style: Lamp-Lamp1-Yellow
    Lamp1 (594,293 53x54), variable: Auto_Cycle_Fix2.Fixture_2.CC3_Output.Work_Position, style: Lamp-Lamp1-Yellow
    Lamp1 (592,361 53x54), variable: Auto_Cycle_Fix2.Fixture_2.CC5_Output.Work_Position, style: Lamp-Lamp1-Yellow
    Textfield (579,178 76x30), "Clamp"
    Lamp1 (709,227 53x54), variable: Auto_Cycle_Fix2.Fixture_2.CC1_Output.Home_Position, style: Lamp-Lamp1-Yellow
    Lamp1 (708,293 53x54), variable: Auto_Cycle_Fix2.Fixture_2.CC3_Output.Home_Position, style: Lamp-Lamp1-Yellow
    Lamp1 (706,361 53x54), variable: Auto_Cycle_Fix2.Fixture_2.CC5_Output.Home_Position, style: Lamp-Lamp1-Yellow
    Textfield (693,178 84x30), "Declamp"
    Textfield (493,443 76x30), "CC2"
    Textfield (492,509 75x30), "CC4"
    Textfield (491,578 73x30), "CC6"
    Lamp1 (594,433 53x54), variable: Auto_Cycle_Fix2.Fixture_2.CC2_Output.Work_Position, style: Lamp-Lamp1-Yellow
    Lamp1 (593,499 53x54), variable: Auto_Cycle_Fix2.Fixture_2.CC4_Output.Work_Position, style: Lamp-Lamp1-Yellow
    Lamp1 (591,567 53x54), variable: Auto_Cycle_Fix2.Fixture_2.CC6_Output.Work_Position, style: Lamp-Lamp1-Yellow
    Lamp1 (708,433 53x54), variable: Auto_Cycle_Fix2.Fixture_2.CC2_Output.Home_Position, style: Lamp-Lamp1-Yellow
    Lamp1 (707,499 53x54), variable: Auto_Cycle_Fix2.Fixture_2.CC4_Output.Home_Position, style: Lamp-Lamp1-Yellow
    Lamp1 (705,567 53x54), variable: Auto_Cycle_Fix2.Fixture_2.CC6_Output.Home_Position, style: Lamp-Lamp1-Yellow
    Button (134,215 112x48)
        p573394764: Auto_Cycle_Fix2.Fixture_2.CC1_Input.Auto_Sel
        toggle Auto_Cycle_Fix2.Fixture_2.CC1_Input.Auto_Sel
    Textfield (33,228 65x30), "CC1"
    Button (133,285 112x48)
        p573394764: Auto_Cycle_Fix2.Fixture_2.CC2_Input.Auto_Sel
        toggle Auto_Cycle_Fix2.Fixture_2.CC2_Input.Auto_Sel
    Textfield (32,298 65x30), "CC2"
    Button (134,356 112x48)
        p573394764: Auto_Cycle_Fix2.Fixture_2.CC3_Input.Auto_Sel
        toggle Auto_Cycle_Fix2.Fixture_2.CC3_Input.Auto_Sel
    Textfield (33,369 65x30), "CC3"
    Button (134,427 112x48)
        p573394764: Auto_Cycle_Fix2.Fixture_2.CC4_Input.Auto_Sel
        toggle Auto_Cycle_Fix2.Fixture_2.CC4_Input.Auto_Sel
    Textfield (33,440 65x30), "CC4"
    Button (134,499 112x48)
        p573394764: Auto_Cycle_Fix2.Fixture_2.CC5_Input.Auto_Sel
        toggle Auto_Cycle_Fix2.Fixture_2.CC5_Input.Auto_Sel
    Textfield (33,512 65x30), "CC5"
    Button (133,571 112x48)
        p573394764: Auto_Cycle_Fix2.Fixture_2.CC6_Input.Auto_Sel
        toggle Auto_Cycle_Fix2.Fixture_2.CC6_Input.Auto_Sel
    Textfield (32,584 65x30), "CC6"
    Button (283,215 112x48)
        p573394764: Auto_Cycle_Fix2.Fixture_2.CC1_Input.Manual_Sel
        toggle Auto_Cycle_Fix2.Fixture_2.CC1_Input.Manual_Sel
    Button (282,285 112x48)
        p573394764: Auto_Cycle_Fix2.Fixture_2.CC2_Input.Manual_Sel
        toggle Auto_Cycle_Fix2.Fixture_2.CC2_Input.Manual_Sel
    Button (283,356 112x48)
        p573394764: Auto_Cycle_Fix2.Fixture_2.CC3_Input.Manual_Sel
        toggle Auto_Cycle_Fix2.Fixture_2.CC3_Input.Manual_Sel
    Button (283,427 112x48)
        p573394764: Auto_Cycle_Fix2.Fixture_2.CC4_Input.Manual_Sel
        toggle Auto_Cycle_Fix2.Fixture_2.CC4_Input.Manual_Sel
    Button (283,499 112x48)
        p573394764: Auto_Cycle_Fix2.Fixture_2.CC5_Input.Manual_Sel
        toggle Auto_Cycle_Fix2.Fixture_2.CC5_Input.Manual_Sel
    Button (282,571 112x48)
        p573394764: Auto_Cycle_Fix2.Fixture_2.CC6_Input.Manual_Sel
        toggle Auto_Cycle_Fix2.Fixture_2.CC6_Input.Manual_Sel
    Textfield (283,156 97x30), "Manual"
END_VISUALIZATION
